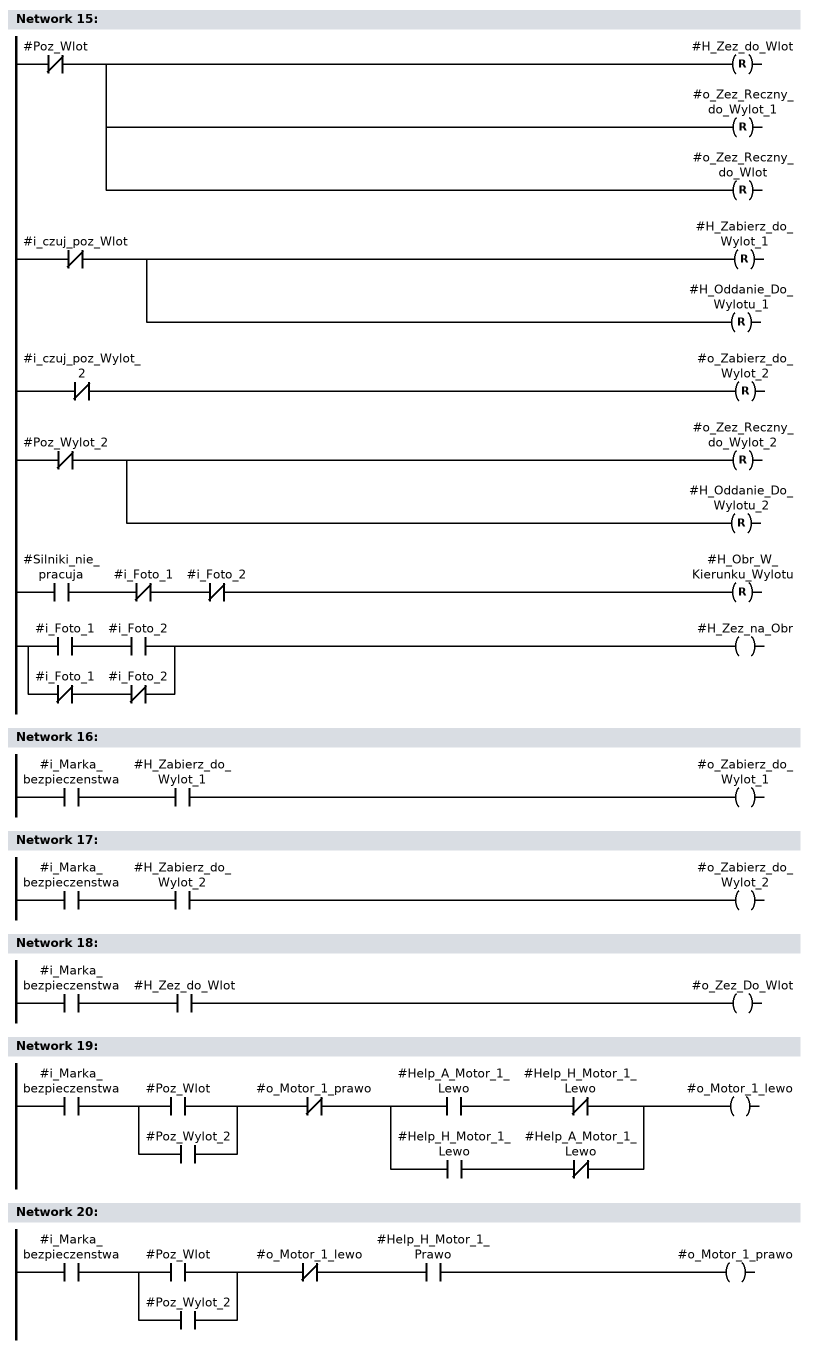
NETWORK
TITLE =
//Warunki skrajne
//
      AN    #Poz_Wlot;
      R     #H_Zez_do_Wlot;
//      R     #H_Zabierz_do_Wylot_1
      R     #o_Zez_Reczny_do_Wylot_1;
      R     #o_Zez_Reczny_do_Wlot;
      AN    #i_czuj_poz_Wlot;
      R     #H_Zabierz_do_Wylot_1;
      R     #H_Oddanie_Do_Wylotu_1;
      AN    #i_czuj_poz_Wylot_2;
      R     #o_Zabierz_do_Wylot_2;
      AN    #Poz_Wylot_2;
//      R     #o_Zabierz_do_Wylot_2
      R     #o_Zez_Reczny_do_Wylot_2;
      R     #H_Oddanie_Do_Wylotu_2;
      A     #Silniki_nie_pracuja;
      AN    #i_Foto_1;
      AN    #i_Foto_2;
      R     #H_Obr_W_Kierunku_Wylotu;
      A     #i_Foto_1;
      A     #i_Foto_2;
      O;
      AN    #i_Foto_1;
      AN    #i_Foto_2;
      =     #H_Zez_na_Obr;
NETWORK
TITLE =
//Sygnal zabierz Wylot_1
      A     #i_Marka_bezpieczenstwa;
      A     #H_Zabierz_do_Wylot_1;
      =     #o_Zabierz_do_Wylot_1;
NETWORK
TITLE =
//Sygnal zabierz Wylot_2
      A     #i_Marka_bezpieczenstwa;
      A     #H_Zabierz_do_Wylot_2;
      =     #o_Zabierz_do_Wylot_2;
NETWORK
TITLE =
//zezwolenie do porzedniej
      A     #i_Marka_bezpieczenstwa;
      A     #H_Zez_do_Wlot;
      =     #o_Zez_Do_Wlot;
NETWORK
TITLE =
////jazda automatyka reczny przod
      A     #i_Marka_bezpieczenstwa;
      A(;
      O     #Poz_Wlot;
      O     #Poz_Wylot_2;
      );
      AN    #o_Motor_1_prawo;
      A(;
      A     #Help_A_Motor_1_Lewo;
      AN    #Help_H_Motor_1_Lewo;
      O;
      A     #Help_H_Motor_1_Lewo;
      AN    #Help_A_Motor_1_Lewo;
      );
      =     #o_Motor_1_lewo;
NETWORK
TITLE =
////Jazda reczny tyl
      A     #i_Marka_bezpieczenstwa;
      A(;
      O     #Poz_Wlot;
      O     #Poz_Wylot_2;
      );
      AN    #o_Motor_1_lewo;
      A     #Help_H_Motor_1_Prawo;
      =     #o_Motor_1_prawo;
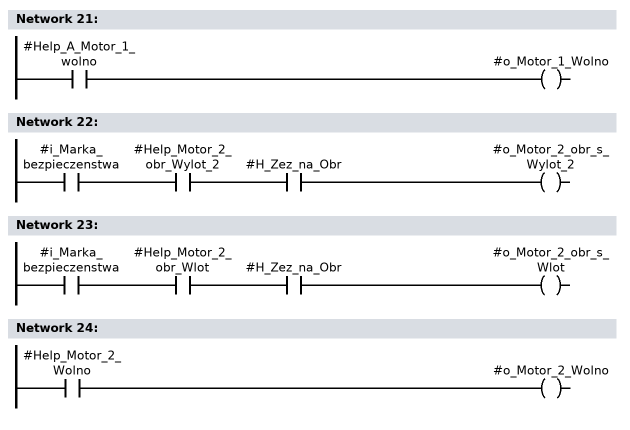
NETWORK
TITLE =
//Motor 1 wolno
      A     #Help_A_Motor_1_wolno;
      =     #o_Motor_1_Wolno;
NETWORK
TITLE =
//obrot obrotnica cc-wise
      A     #i_Marka_bezpieczenstwa;
      A     #Help_Motor_2_obr_Wylot_2;
      A     #H_Zez_na_Obr;
      =     #o_Motor_2_obr_s_Wylot_2;
NETWORK
TITLE =
//obrot obrotnica c-wise
      A     #i_Marka_bezpieczenstwa;
      A     #Help_Motor_2_obr_Wlot;
      A     #H_Zez_na_Obr;
      =     #o_Motor_2_obr_s_Wlot;
NETWORK
TITLE =
//motor 2 wolno
      A     #Help_Motor_2_Wolno;
      =     #o_Motor_2_Wolno;
END_FUNCTION_BLOCK

FUNCTION_BLOCK "Banda_Poj_+_Winda"	// FB 37
//Funkcja realizujaca koncepcje bandy pojedycznej, ktora uwzglednia rowniez tryb 
//reczny. W celu lepszego sterowania trybem recznym nalezy do³o¿yæ:
//-fotokomorki na tyle bandy.
//-fotokomorka na tyle okresla rowniez zajetosc
//-jazda do tylu bandy mozliwa
//-jazda do przodu poza fotokomorke mozliwa gdy nastepna w ruchu i wolna.
//-do³o¿enie okresnia trybu reczny/auto gdzie auto to 1 
//
//
//Do wersji z winda
//-winda rowniez aktywna gdy dojechala do gory tkz nadrabianie wysokosci
//-uwzglednione dwa czujniki od skrajnych pozycji windy
//-banda poprzedzajaca poziom 0
//-banda nastepna poziom +1
//
AUTHOR : Kng
FAMILY : Bandy
NAME : B_Single
VERSION : 0.0
VAR_INPUT
  i_Marka_Bezpieczenstwa : BOOL ;
  i_Blokada_Gdy_Uzbrajanie : BOOL ;	//Sygnal Rezerwy
  i_Auto_Reczny : BOOL ;	//1-auto,0-reczny
  i_Foto_Przod : BOOL ;	//Foto na koncu tasmy
  i_Foto_Tyl : BOOL ;	//Foto zapobiegajace wyjechaniu palety do tylu
  i_Winda_W_Gorze : BOOL ;
  i_Winda_W_Dole : BOOL ;
  i_Zez_Od_Nast : BOOL ;
  i_Paleta_Dost_Od_Nast : BOOL ;
  i_Zez_Reczny_Od_Nast : BOOL ;
  i_Zabierz_Od_Pop : BOOL ;
  i_Zez_Reczny_Od_Pop : BOOL ;
  i_PB_Jazda_Tyl : BOOL ;
  i_PB_Jazda_Przod : BOOL ;
  i_PB_Winda_Gora : BOOL ;
  i_PB_Winda_Dol : BOOL ;
  Czas_Kontroli_Przejazdu : TIME ;
END_VAR
VAR_OUTPUT
  o_Zabierz_Do_Nast : BOOL ;	//Rozkaz pobrania do nast bandy
  o_Zez_Do_Pop : BOOL ;
  o_Paleta_Dost_Do_Pop : BOOL ;
  o_Motor_Lewo : BOOL ;
  o_Motor_Prawo : BOOL ;
  o_Winda_Gora : BOOL ;
  o_Winda_Dol : BOOL ;
  o_Zez_Reczny_Do_Nast : BOOL ;
  o_Zez_Reczny_Do_Pop : BOOL ;
  o_Zajetosc_Nieb : BOOL ;	//Dla bezpieczenstwa transportu
  o_Paleta_Na_Stanowisku : BOOL ;	//Informacja o tym ze paleta jest na stanowisku
END_VAR
VAR
  Czas_kontrolny : FB 21;
  Czas_Windy : SFB 4;
  Help_A_Motor_Lewo : BOOL ;
  S_Help_Zab_Od_Pop : BOOL ;
  Stop_Czas_Kontrolny : BOOL ;
  Zbocze_1 : BOOL ;
  Zbocze_2 : BOOL ;
  Blokada_Wjazdu : BOOL ;
  Help_H_Motor_Prawo : BOOL ;
  Help_H_Motor_Lewo : BOOL ;
  Toggle : BOOL ;	//bit przemienny dla auto i hand
  H_Winda_A_Gora : BOOL ;
  H_Winda_A_Dol : BOOL ;
  H_Kontr_Windy_Gora : BOOL ;	//Kontrola by winda nie opadala
  H_Kontr_Windy_Dol : BOOL ;
  H_Winda_H_Gora : BOOL ;
  H_Winda_H_Dol : BOOL ;
  Czas_Opoz_Windy : SFB 4;
END_VAR
VAR_TEMP
  Temp_Help_1 : BOOL ;
  Temp_Help_2 : BOOL ;
  Czas_zadany : TIME ;
  Czas_aktualny : TIME ;
END_VAR
BEGIN
NETWORK
TITLE =
//
// B1        B2         foto_1    foto_2         B5        B6
//(\\\\\\\\\\\\\\\\\\)  (\\\\\\\\\\\\\\\\\\)  (\\\\\\\\\\\\\\\\\\)
//                  M1                    M2                     M3
//         
//        zabierz <-- pobierz      |  zabierz    <--  pobierz  
//     zez_do_pop --> zez_od_nast  |  zez_od_pop -->  zez_od_nast
//                                  
//-Uklad dzielony jest na realizowane funkcje
//
//         <----------------------------------------- kierunek
//                  
//
// ten network celowo jest pusty
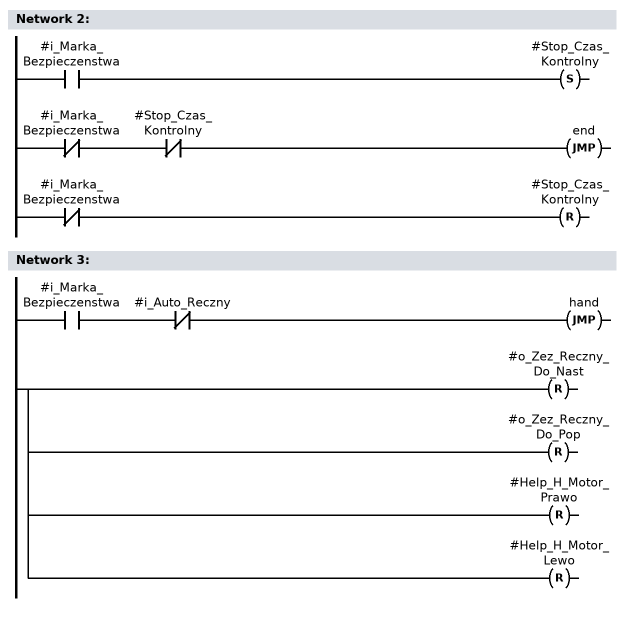
NETWORK
TITLE =
//Sprawdzenie stanu bezpieczenstwa lub freeze
//Skocz jezeli brak marki bezpieczenstwa
//Marka bezpieczenstwa ok gdy wysoki
      A     #i_Marka_Bezpieczenstwa;
      S     #Stop_Czas_Kontrolny;
      AN    #i_Marka_Bezpieczenstwa;
      AN    #Stop_Czas_Kontrolny;
      JC    end;
      AN    #i_Marka_Bezpieczenstwa;
      R     #Stop_Czas_Kontrolny;
NETWORK
TITLE =
//Wyznczenie zbocza pozytywnego i negatywnego
//skok do trybu recznego 
      A     #i_Marka_Bezpieczenstwa;
      AN    #i_Auto_Reczny;
      JC    hand;
//czyszczenie trybu recznego
      SET;
      R     #o_Zez_Reczny_Do_Nast;
      R     #o_Zez_Reczny_Do_Pop;
      R     #Help_H_Motor_Prawo;
      R     #Help_H_Motor_Lewo;
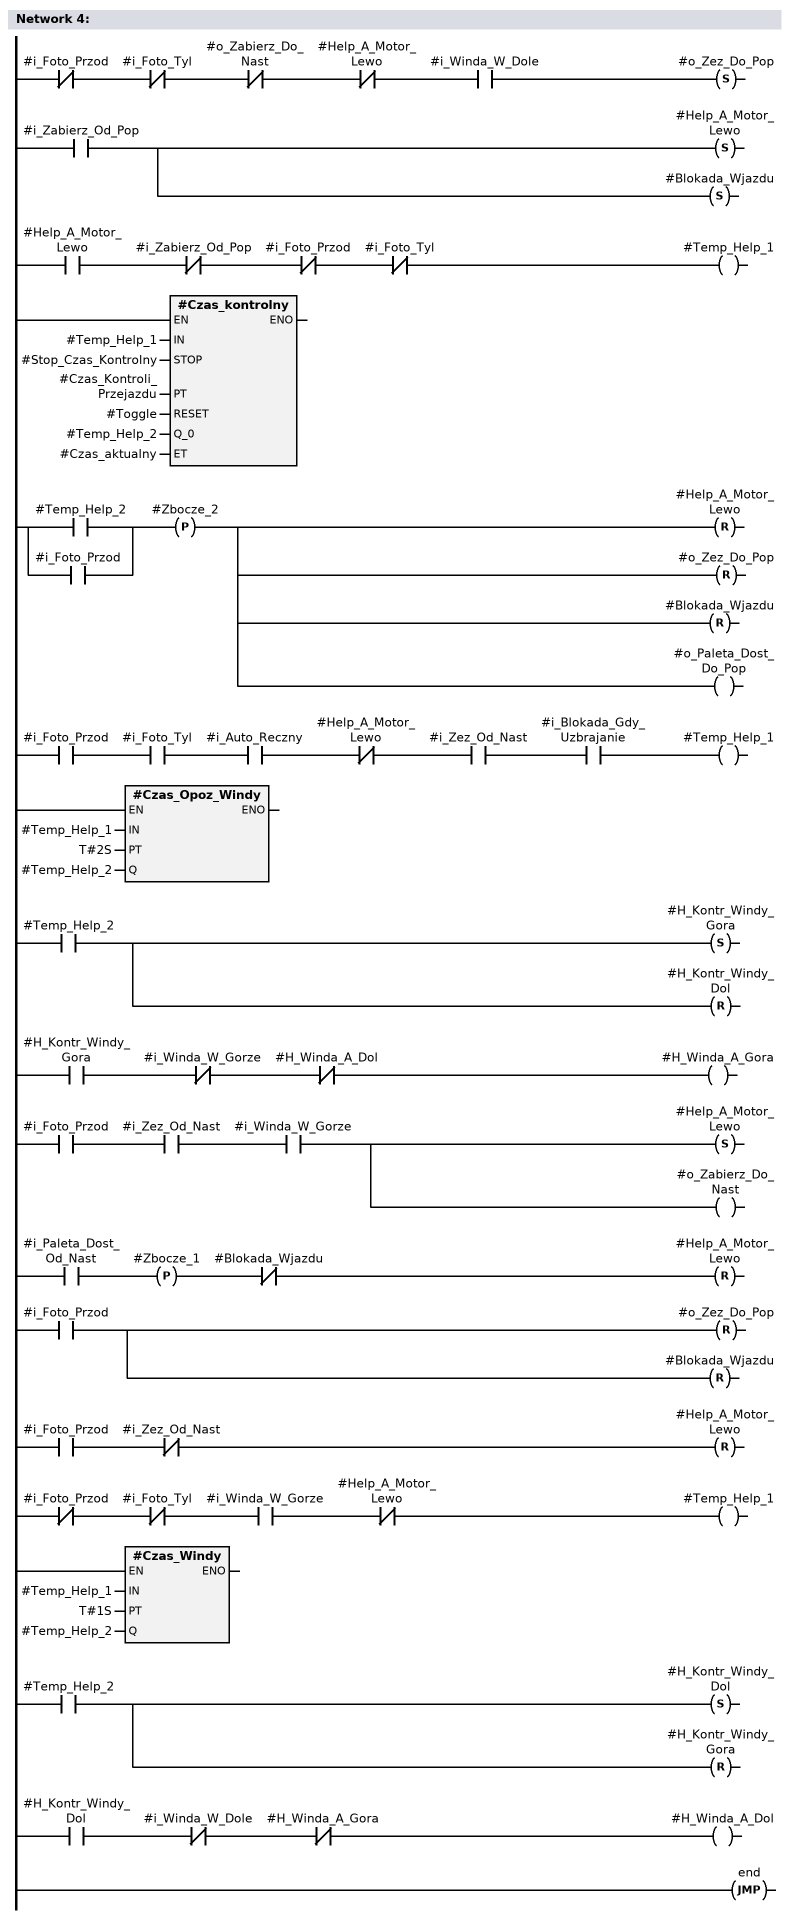
NETWORK
TITLE =
//Banda pusta zezwol na wjazd
      AN    #i_Foto_Przod;
      AN    #i_Foto_Tyl;	//dodano bo hand
      AN    #o_Zabierz_Do_Nast;
      AN    #Help_A_Motor_Lewo;
      A     #i_Winda_W_Dole;
      S     #o_Zez_Do_Pop;
      A     #i_Zabierz_Od_Pop;
      S     #Help_A_Motor_Lewo;
      S     #Blokada_Wjazdu;
//Warunek gdy pobranie z poprzedniej i miejsce foto srodek
//jest zajete
      A     #Help_A_Motor_Lewo;
      AN    #i_Zabierz_Od_Pop;
      AN    #i_Foto_Przod;
      AN    #i_Foto_Tyl;	//dodano bo hand
      =     #Temp_Help_1;
      CALL  #Czas_kontrolny (
           IN                       := #Temp_Help_1,
           STOP                     := #Stop_Czas_Kontrolny,
           PT                       := #Czas_Kontroli_Przejazdu,
           RESET                    := #Toggle,
           Q_0                      := #Temp_Help_2,
           ET                       := #Czas_aktualny);
//Paleta dostarczona
      A     #Temp_Help_2;
      O;
      A     #i_Foto_Przod;
      FP    #Zbocze_2;
      R     #Help_A_Motor_Lewo;
      R     #o_Zez_Do_Pop;
      R     #Blokada_Wjazdu;
      =     #o_Paleta_Dost_Do_Pop;
//Podniesiesnie plety na poziom +1
      A     #i_Foto_Przod;
      A     #i_Foto_Tyl;	//Aby bylo pewne pokrycie
      A     #i_Auto_Reczny;
      AN    #Help_A_Motor_Lewo;
      A     #i_Zez_Od_Nast;
      A     #i_Blokada_Gdy_Uzbrajanie;
      =     #Temp_Help_1;
      CALL  #Czas_Opoz_Windy (
           IN                       := #Temp_Help_1,
           PT                       := T#2S,
           Q                        := #Temp_Help_2);
      A     #Temp_Help_2;
      S     #H_Kontr_Windy_Gora;
      R     #H_Kontr_Windy_Dol;
      A     #H_Kontr_Windy_Gora;
//Wylaczenie windy gdy znajduje sie w gorze
      AN    #i_Winda_W_Gorze;
      AN    #H_Winda_A_Dol;
      =     #H_Winda_A_Gora;
      A     #i_Foto_Przod;
//jest zezwolenie od nastepnej
      A     #i_Zez_Od_Nast;
      A     #i_Winda_W_Gorze;
      S     #Help_A_Motor_Lewo;
      =     #o_Zabierz_Do_Nast;
      A     #i_Paleta_Dost_Od_Nast;
//Potwierdzenie otrzymania palety
      FP    #Zbocze_1;
      AN    #Blokada_Wjazdu;
      R     #Help_A_Motor_Lewo;
      A     #i_Foto_Przod;
//Gdy zajete Foto_1 brak zezwolenia do poprzedniej
      R     #o_Zez_Do_Pop;
      R     #Blokada_Wjazdu;
      A     #i_Foto_Przod;
//warunkowe zakonczenie pracy silnika gdy brak zezwolenia
//z nastepnej
      AN    #i_Zez_Od_Nast;
      R     #Help_A_Motor_Lewo;
      AN    #i_Foto_Przod;
//Powrot windy na dol
      AN    #i_Foto_Tyl;
      A     #i_Winda_W_Gorze;
      AN    #Help_A_Motor_Lewo;
      =     #Temp_Help_1;
      CALL  #Czas_Windy (
           IN                       := #Temp_Help_1,
           PT                       := T#1S,
           Q                        := #Temp_Help_2);
      A     #Temp_Help_2;
      S     #H_Kontr_Windy_Dol;
      R     #H_Kontr_Windy_Gora;
      A     #H_Kontr_Windy_Dol;
      AN    #i_Winda_W_Dole;
      AN    #H_Winda_A_Gora;
      =     #H_Winda_A_Dol;
      JU    end;
//skocz do koniec
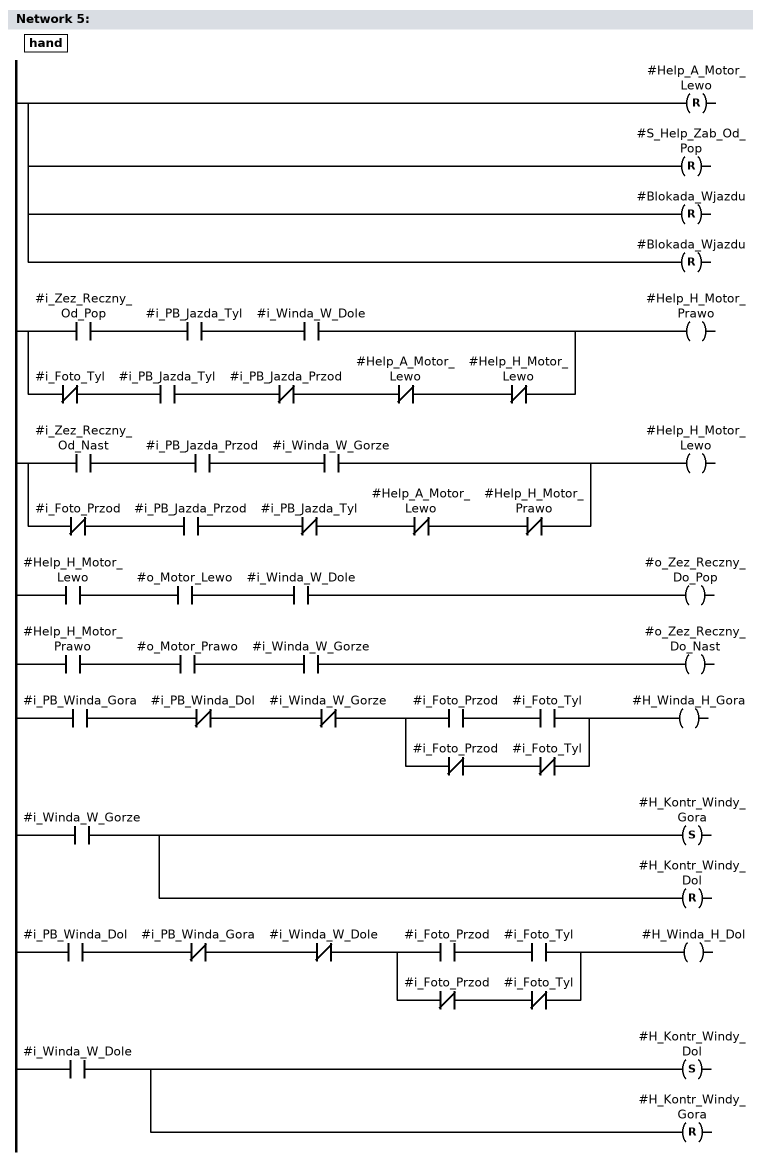
NETWORK
TITLE =
//Tryb reczny
//
hand: NOP   0;
//czyszczenie bitow z automatyki
      SET;
      R     #Help_A_Motor_Lewo;
      R     #S_Help_Zab_Od_Pop;
      R     #Blokada_Wjazdu;
      R     #Blokada_Wjazdu;
//ustawienie przyciskow
//jazda do tylu przycisk tyl
      A     #i_Zez_Reczny_Od_Pop;
      A     #i_PB_Jazda_Tyl;
      A     #i_Winda_W_Dole;
      O;
      AN    #i_Foto_Tyl;
      A(;
      A     #i_PB_Jazda_Tyl;
      AN    #i_PB_Jazda_Przod;
      AN    #Help_A_Motor_Lewo;
      AN    #Help_H_Motor_Lewo;
      );
      =     #Help_H_Motor_Prawo;
//jazda do przodu
      A     #i_Zez_Reczny_Od_Nast;
      A     #i_PB_Jazda_Przod;
      A     #i_Winda_W_Gorze;
      O;
      AN    #i_Foto_Przod;
      A(;
      A     #i_PB_Jazda_Przod;
      AN    #i_PB_Jazda_Tyl;
      AN    #Help_A_Motor_Lewo;
      AN    #Help_H_Motor_Prawo;
      );
      =     #Help_H_Motor_Lewo;
//zezwolenie do poprzedniej
      A     #Help_H_Motor_Lewo;
      A     #o_Motor_Lewo;
      A     #i_Winda_W_Dole;
      =     #o_Zez_Reczny_Do_Pop;
//zezwolenie do nastepnej
      A     #Help_H_Motor_Prawo;
      A     #o_Motor_Prawo;
      A     #i_Winda_W_Gorze;
      =     #o_Zez_Reczny_Do_Nast;
//Jazda windy   gora
      A     #i_PB_Winda_Gora;
      AN    #i_PB_Winda_Dol;
      AN    #i_Winda_W_Gorze;
      A(;
      A     #i_Foto_Przod;
      A     #i_Foto_Tyl;
      O;
      AN    #i_Foto_Przod;
      AN    #i_Foto_Tyl;
      );
      =     #H_Winda_H_Gora;
      A     #i_Winda_W_Gorze;
      S     #H_Kontr_Windy_Gora;
      R     #H_Kontr_Windy_Dol;
//Jazda Windy dol
      A     #i_PB_Winda_Dol;
      AN    #i_PB_Winda_Gora;
      AN    #i_Winda_W_Dole;
      A(;
      A     #i_Foto_Przod;
      A     #i_Foto_Tyl;
      O;
      AN    #i_Foto_Przod;
      AN    #i_Foto_Tyl;
      );
      =     #H_Winda_H_Dol;
      A     #i_Winda_W_Dole;
      S     #H_Kontr_Windy_Dol;
      R     #H_Kontr_Windy_Gora;
NETWORK
TITLE =
//Przypisanie wyjsc
//Koniec skoku
end:  NOP   0;
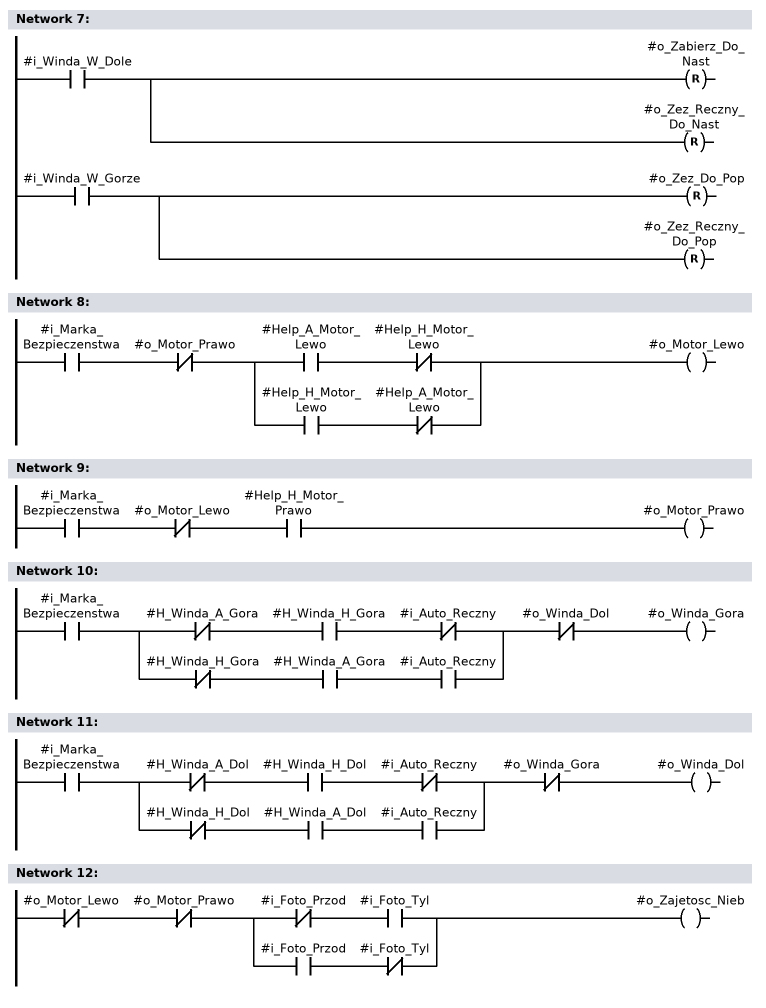
NETWORK
TITLE =
//warunki skrajne
//
      A     #i_Winda_W_Dole;
      R     #o_Zabierz_Do_Nast;
      R     #o_Zez_Reczny_Do_Nast;
      A     #i_Winda_W_Gorze;
      R     #o_Zez_Do_Pop;
      R     #o_Zez_Reczny_Do_Pop;
NETWORK
TITLE =
////jazda automatyka reczny przod
      A     #i_Marka_Bezpieczenstwa;
      AN    #o_Motor_Prawo;
      A(;
      A     #Help_A_Motor_Lewo;
      AN    #Help_H_Motor_Lewo;
      O;
      A     #Help_H_Motor_Lewo;
      AN    #Help_A_Motor_Lewo;
      );
      =     #o_Motor_Lewo;
NETWORK
TITLE =
////Jazda reczny tyl
      A     #i_Marka_Bezpieczenstwa;
      AN    #o_Motor_Lewo;
      A     #Help_H_Motor_Prawo;
      =     #o_Motor_Prawo;
NETWORK
TITLE =
//winda gora
//
      A     #i_Marka_Bezpieczenstwa;
      A(;
      AN    #H_Winda_A_Gora;
      A     #H_Winda_H_Gora;
      AN    #i_Auto_Reczny;
      O;
      AN    #H_Winda_H_Gora;
      A     #H_Winda_A_Gora;
      A     #i_Auto_Reczny;
      );
      AN    #o_Winda_Dol;
      =     #o_Winda_Gora;
NETWORK
TITLE =
//winda dol
      A     #i_Marka_Bezpieczenstwa;
      A(;
      AN    #H_Winda_A_Dol;
      A     #H_Winda_H_Dol;
      AN    #i_Auto_Reczny;
      O;
      AN    #H_Winda_H_Dol;
      A     #H_Winda_A_Dol;
      A     #i_Auto_Reczny;
      );
      AN    #o_Winda_Gora;
      =     #o_Winda_Dol;
NETWORK
TITLE =
//Zajetosc
      AN    #o_Motor_Lewo;
      AN    #o_Motor_Prawo;
      A(;
      AN    #i_Foto_Przod;
      A     #i_Foto_Tyl;
      O;
      A     #i_Foto_Przod;
      AN    #i_Foto_Tyl;
      );
      =     #o_Zajetosc_Nieb;
NETWORK
TITLE =
//Koniec
//koniec
      BEU;
END_FUNCTION_BLOCK

FUNCTION_BLOCK "Obr_Na_Poz_1_Pelny"	// FB 61
AUTHOR : Kng
NAME : B_Obr
VERSION : 0.1
VAR_INPUT
  i_Auto_Reczny : BOOL ;
  i_Tryb_Uzbrajanie : BOOL ;	//Tryb uzbrajania palaty (mozliwosci pelnego obrotu)
  i_Obracaj_W_Lewo : BOOL ;	//Aktywne tylko w trybie uzbrajania
  i_Obracaj_W_Prawo : BOOL ;	//Aktywne tylko w trybie uzbrajania
  i_Jedz_Na_0st : BOOL ;
  i_Jedz_Na_90st : BOOL ;
  i_Czujnik_0st : BOOL ;
  i_Czujnik_90st : BOOL ;
  i_Czujnik_Ham_0st : BOOL ;
  i_Czujnik_Ham_90st : BOOL ;
  i_Odblokuj_Obrotnice : BOOL ;
END_VAR
VAR_OUTPUT
  o_Na_Pozycji_0st : BOOL ;	//Obrotnica na pozycji 0 stopni
  o_Na_Pozycji_90st : BOOL ;	//Obrotnica na pozycji 90 stopni
  o_Motor_Wolno : BOOL ;
  o_Odblokowanie_Rolek : BOOL ;
  o_Uzbrajanie : BOOL ;
END_VAR
VAR_IN_OUT
  io_Talerz_w_Lewo : BOOL ;
  io_Talerz_w_Prawo : BOOL ;
END_VAR
VAR
  Czas_Dojscia : SFB 4;
  Czas_Startu : SFB 4;
  Help_Start : BOOL ;
  H_Blokada_Uzbrajania : BOOL ;
  H_2 : BOOL ;
  H_3 : BOOL ;
  H_4 : BOOL ;
END_VAR
VAR_TEMP
  Help_1 : BOOL ;
END_VAR
BEGIN
NETWORK
TITLE =
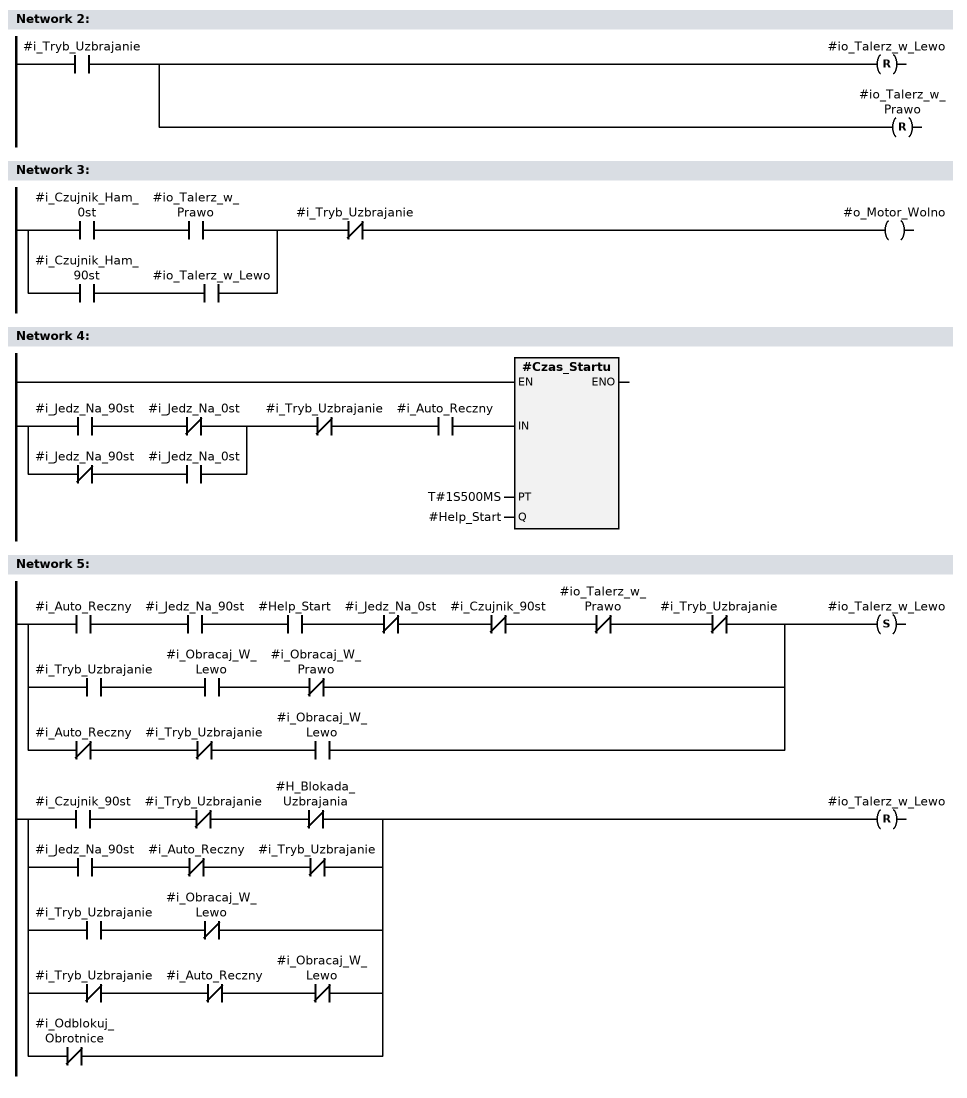
NETWORK
TITLE =
//Tryb uzbrajania resetuje wszystkie bity
      A     #i_Tryb_Uzbrajanie;
      R     #io_Talerz_w_Lewo;
      R     #io_Talerz_w_Prawo;
NETWORK
TITLE =
//Motor wolno gdy czujniki hamowania
      A(;
      A     #i_Czujnik_Ham_0st;
      A     #io_Talerz_w_Prawo;
      O;
      A     #i_Czujnik_Ham_90st;
      A     #io_Talerz_w_Lewo;
      );
      AN    #i_Tryb_Uzbrajanie;
      =     #o_Motor_Wolno;
NETWORK
TITLE =
      A(;
      A     #i_Jedz_Na_90st;
      AN    #i_Jedz_Na_0st;
      O;
      AN    #i_Jedz_Na_90st;
      A     #i_Jedz_Na_0st;
      );
      AN    #i_Tryb_Uzbrajanie;
      A     #i_Auto_Reczny;
      =     L 1.0;
      BLD   103;
      CALL  #Czas_Startu (
           IN                       := L 1.0,
           PT                       := T#1S500MS,
           Q                        := #Help_Start);
      NOP   0;
NETWORK
TITLE =
      A(;
      A     #i_Auto_Reczny;
      A     #i_Jedz_Na_90st;
      A     #Help_Start;
      AN    #i_Jedz_Na_0st;
      AN    #i_Czujnik_90st;
      AN    #io_Talerz_w_Prawo;
      AN    #i_Tryb_Uzbrajanie;
      O;
      A     #i_Tryb_Uzbrajanie;
      A     #i_Obracaj_W_Lewo;
      AN    #i_Obracaj_W_Prawo;
      O;
      AN    #i_Auto_Reczny;
      AN    #i_Tryb_Uzbrajanie;
      A     #i_Obracaj_W_Lewo;
      );
      S     #io_Talerz_w_Lewo;
      A(;
      A     #i_Czujnik_90st;
      AN    #i_Tryb_Uzbrajanie;
      AN    #H_Blokada_Uzbrajania;
      O;
      A     #i_Jedz_Na_90st;
      AN    #i_Auto_Reczny;
      AN    #i_Tryb_Uzbrajanie;
      O;
      A     #i_Tryb_Uzbrajanie;
      AN    #i_Obracaj_W_Lewo;
      O;
      AN    #i_Tryb_Uzbrajanie;
      AN    #i_Auto_Reczny;
      AN    #i_Obracaj_W_Lewo;
      ON    #i_Odblokuj_Obrotnice;
      );
      R     #io_Talerz_w_Lewo;
      NOP   0;
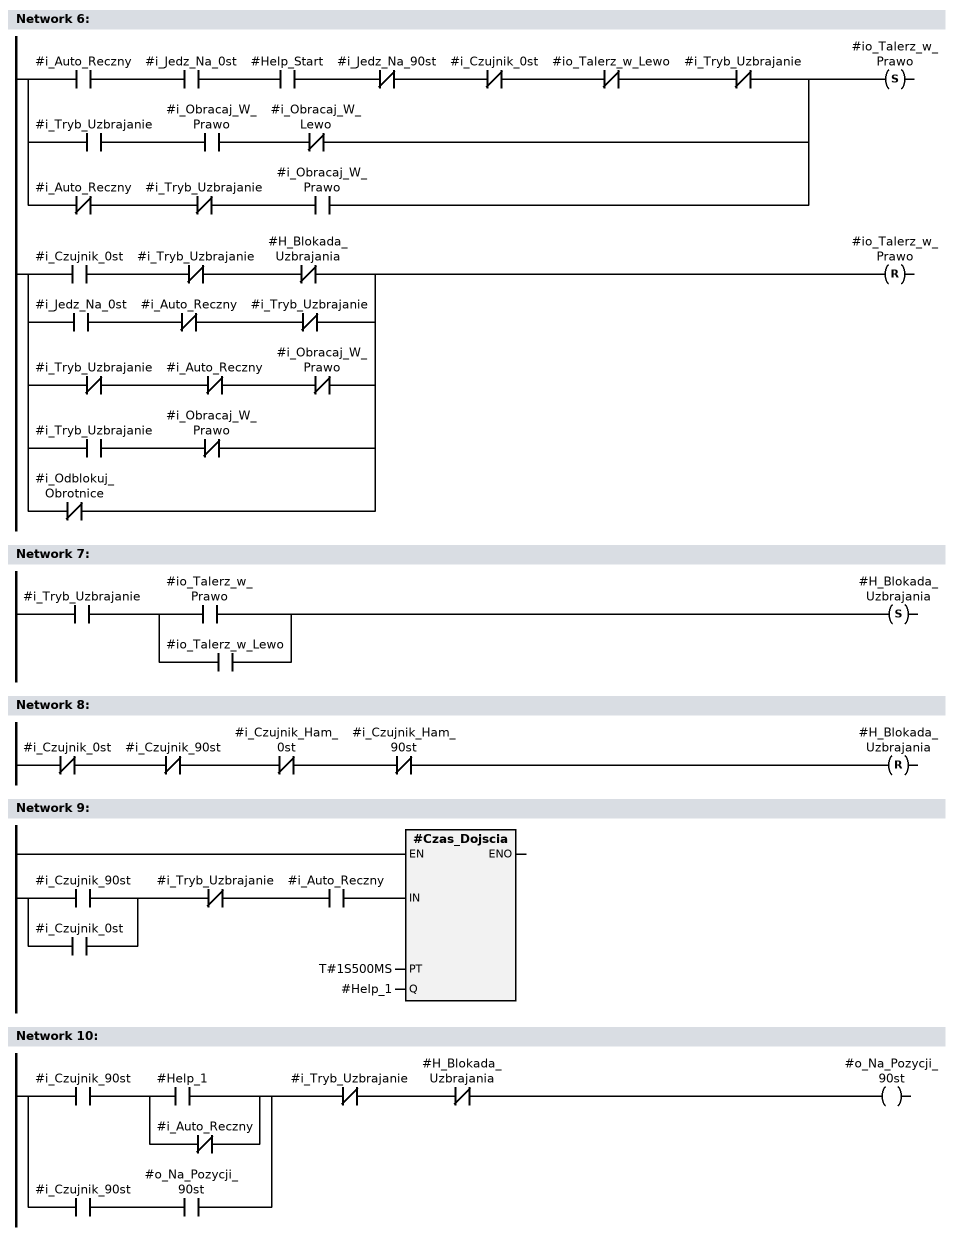
NETWORK
TITLE =
      A(;
      A     #i_Auto_Reczny;
      A     #i_Jedz_Na_0st;
      A     #Help_Start;
      AN    #i_Jedz_Na_90st;
      AN    #i_Czujnik_0st;
      AN    #io_Talerz_w_Lewo;
      AN    #i_Tryb_Uzbrajanie;
      O;
      A     #i_Tryb_Uzbrajanie;
      A     #i_Obracaj_W_Prawo;
      AN    #i_Obracaj_W_Lewo;
      O;
      AN    #i_Auto_Reczny;
      AN    #i_Tryb_Uzbrajanie;
      A     #i_Obracaj_W_Prawo;
      );
      S     #io_Talerz_w_Prawo;
      A(;
      A     #i_Czujnik_0st;
      AN    #i_Tryb_Uzbrajanie;
      AN    #H_Blokada_Uzbrajania;
      O;
      A     #i_Jedz_Na_0st;
      AN    #i_Auto_Reczny;
      AN    #i_Tryb_Uzbrajanie;
      O;
      AN    #i_Tryb_Uzbrajanie;
      AN    #i_Auto_Reczny;
      AN    #i_Obracaj_W_Prawo;
      O;
      A     #i_Tryb_Uzbrajanie;
      AN    #i_Obracaj_W_Prawo;
      ON    #i_Odblokuj_Obrotnice;
      );
      R     #io_Talerz_w_Prawo;
      NOP   0;
NETWORK
TITLE =
//Jezeli byl tryb uzbrajania aktywny i nastapil przejazd aktywuj h_1
      A     #i_Tryb_Uzbrajanie;
      A(;
      O     #io_Talerz_w_Prawo;
      O     #io_Talerz_w_Lewo;
      );
      S     #H_Blokada_Uzbrajania;
NETWORK
TITLE =
//Reset blokady uzbrajania
      AN    #i_Czujnik_0st;
      AN    #i_Czujnik_90st;
      AN    #i_Czujnik_Ham_0st;
      AN    #i_Czujnik_Ham_90st;
      R     #H_Blokada_Uzbrajania;
NETWORK
TITLE =
      A(;
      O     #i_Czujnik_90st;
      O     #i_Czujnik_0st;
      );
      AN    #i_Tryb_Uzbrajanie;
      A     #i_Auto_Reczny;
      =     L 1.0;
      BLD   103;
      CALL  #Czas_Dojscia (
           IN                       := L 1.0,
           PT                       := T#1S500MS,
           Q                        := #Help_1);
      NOP   0;
NETWORK
TITLE =
      A(;
      A     #i_Czujnik_90st;
      A(;
      O     #Help_1;
      ON    #i_Auto_Reczny;
      );
      O;
      A     #i_Czujnik_90st;
      A     #o_Na_Pozycji_90st;
      );
      AN    #i_Tryb_Uzbrajanie;
      AN    #H_Blokada_Uzbrajania;
      =     #o_Na_Pozycji_90st;
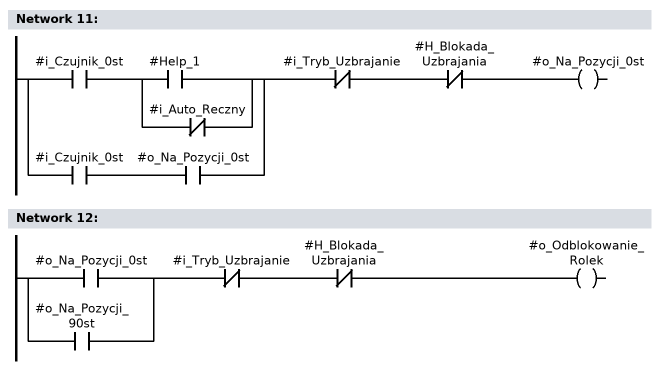
NETWORK
TITLE =
      A(;
      A     #i_Czujnik_0st;
      A(;
      O     #Help_1;
      ON    #i_Auto_Reczny;
      );
      O;
      A     #i_Czujnik_0st;
      A     #o_Na_Pozycji_0st;
      );
      AN    #i_Tryb_Uzbrajanie;
      AN    #H_Blokada_Uzbrajania;
      =     #o_Na_Pozycji_0st;
NETWORK
TITLE =
//Odblokowanie napedu rolkowego
      A(;
      O     #o_Na_Pozycji_0st;
      O     #o_Na_Pozycji_90st;
      );
      AN    #i_Tryb_Uzbrajanie;
      AN    #H_Blokada_Uzbrajania;
      =     #o_Odblokowanie_Rolek;
END_FUNCTION_BLOCK

FUNCTION "Funkcja_Bezpieczenstwa" : VOID	// FC 3
VERSION : 0.1
VAR_TEMP
  Temp_Help_1 : BOOL ;
  Temp_Help_2 : BOOL ;
END_VAR
BEGIN
NETWORK
TITLE =
//Ten network celowo jest wolny
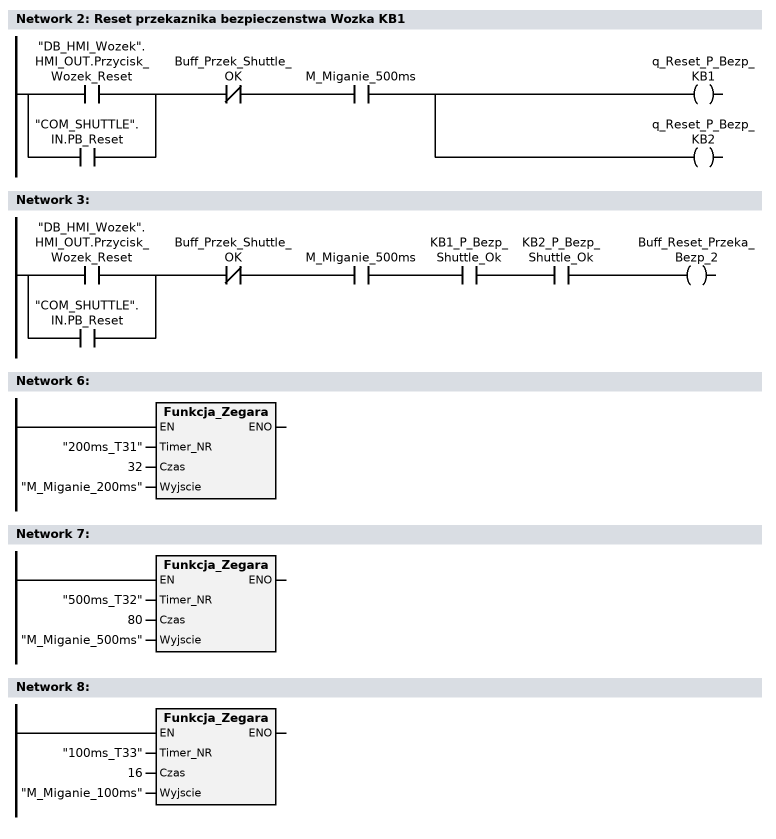
NETWORK
TITLE = Reset przekaznika bezpieczenstwa Wozka KB1
//Reset przekaznikow bezpieczenstwa stanowisk KB1,KB2
      A(;
      O     "DB_HMI_Wozek".HMI_OUT.Przycisk_Wozek_Reset;
      O     "COM_SHUTTLE".IN.PB_Reset;
      );
      AN    "Buff_Przek_Shuttle_OK";
      A     "M_Miganie_500ms";
      =     "q_Reset_P_Bezp_KB1";
      =     "q_Reset_P_Bezp_KB2";
NETWORK
TITLE =
//Reset przekaznik bezpieczenstwa wozek
      A(;
      O     "DB_HMI_Wozek".HMI_OUT.Przycisk_Wozek_Reset;
      O     "COM_SHUTTLE".IN.PB_Reset;
      );
      AN    "Buff_Przek_Shuttle_OK";
      A     "M_Miganie_500ms";
      A     "KB1_P_Bezp_Shuttle_Ok";
      A     "KB2_P_Bezp_Shuttle_Ok";
      =     "Buff_Reset_Przeka_Bezp_2";
NETWORK
TITLE =
NETWORK
TITLE =
//Zalaczenie szynoprzewodu
      A     "i_Buff_PB_Zal_Wozka";
      L     S5T#1S;
      SD    "Buff_T35";
//----
      A     "Buff_T35";
      FP    "Help_M302.7";
      X     "q_Buff_Zal_Wozka";
      =     "q_Buff_Zal_Wozka";
NETWORK
TITLE =
//Timmer generujacy takt 200ms
//
      CALL  "Funkcja_Zegara" (
           Timer_NR                 := "200ms_T31",
           Czas                     := 32,
           Wyjscie                  := "M_Miganie_200ms");
      NOP   0;
NETWORK
TITLE =
//Timmer generujacy takt 500ms
      CALL  "Funkcja_Zegara" (
           Timer_NR                 := "500ms_T32",
           Czas                     := 80,
           Wyjscie                  := "M_Miganie_500ms");
      NOP   0;
NETWORK
TITLE =
//Timmer generujacy takt 100ms
      CALL  "Funkcja_Zegara" (
           Timer_NR                 := "100ms_T33",
           Czas                     := 16,
           Wyjscie                  := "M_Miganie_100ms");
      NOP   0;
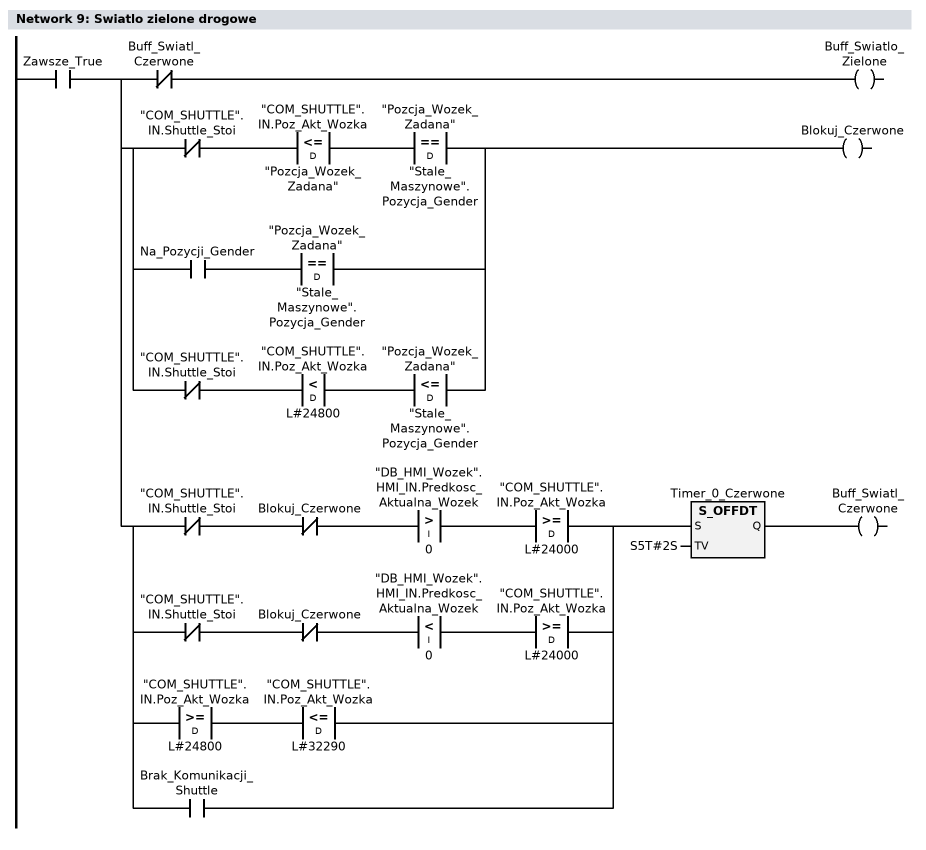
NETWORK
TITLE = Swiatlo zielone drogowe
//Ruch drogowy
//0______24000
//0______26300
//26200__32290
      A     "Zawsze_True";
      =     L 1.0;
      A     L 1.0;
      AN    "Buff_Swiatl_Czerwone";
      =     "Buff_Swiatlo_Zielone";
      A     L 1.0;
      A(;
      AN    "COM_SHUTTLE".IN.Shuttle_Stoi;
      A(;
      L     "COM_SHUTTLE".IN.Poz_Akt_Wozka;
      L     "Pozcja_Wozek_Zadana";
      <=D;
      );
      A(;
      L     "Pozcja_Wozek_Zadana";
      L     "Stale_Maszynowe".Pozycja_Gender;
      ==D;
      );
      O;
      A     "Na_Pozycji_Gender";
      A(;
      L     "Pozcja_Wozek_Zadana";
      L     "Stale_Maszynowe".Pozycja_Gender;
      ==D;
      );
      O;
      AN    "COM_SHUTTLE".IN.Shuttle_Stoi;
      A(;
      L     "COM_SHUTTLE".IN.Poz_Akt_Wozka;
      L     L#24800;
      <D;
      );
      A(;
      L     "Pozcja_Wozek_Zadana";
      L     "Stale_Maszynowe".Pozycja_Gender;
      <=D;
      );
      );
      =     "Blokuj_Czerwone";
      A     L 1.0;
      A(;
      AN    "COM_SHUTTLE".IN.Shuttle_Stoi;
      AN    "Blokuj_Czerwone";
      A(;
      L     "DB_HMI_Wozek".HMI_IN.Predkosc_Aktualna_Wozek;
      L     0;
      >I;
      );
      A(;
      L     "COM_SHUTTLE".IN.Poz_Akt_Wozka;
      L     L#24000;
      >=D;
      );
      O;
      AN    "COM_SHUTTLE".IN.Shuttle_Stoi;
      AN    "Blokuj_Czerwone";
      A(;
      L     "DB_HMI_Wozek".HMI_IN.Predkosc_Aktualna_Wozek;
      L     0;
      <I;
      );
      A(;
      L     "COM_SHUTTLE".IN.Poz_Akt_Wozka;
      L     L#24000;
      >=D;
      );
      O;
      A(;
      L     "COM_SHUTTLE".IN.Poz_Akt_Wozka;
      L     L#24800;
      >=D;
      );
      A(;
      L     "COM_SHUTTLE".IN.Poz_Akt_Wozka;
      L     L#32290;
      <=D;
      );
      O     "Brak_Komunikacji_Shuttle";
      );
      L     S5T#2S;
      SF    "Timer_0_Czerwone";
      NOP   0;
      NOP   0;
      NOP   0;
      A     "Timer_0_Czerwone";
      =     "Buff_Swiatl_Czerwone";
END_FUNCTION

FUNCTION "Wozek_Jezdny_Jazda_2" : VOID	// FC 6
//Funkcja odpowiada za sterowanie ruchem wozka. Uzywa marek od m600.0
AUTHOR : Kng
NAME : Main
VERSION : 0.1
BEGIN
NETWORK
TITLE =
//Ten Network Celowo jest wolny
NETWORK
TITLE =
      CALL  "Wozek_Jezdny_Kolejka";
      NOP   0;
NETWORK
TITLE =
//Sprawdzenie okna dla KB2
      CALL  "Sprawdzenie_Okna" (
           War_Pozycji_Aktualnej    := "COM_SHUTTLE".IN.Poz_Akt_Wozka,
           War_Pozycji_Zadanej      := "COM_SHUTTLE".OUT.Pozycja_Zadana,
           War_Pozycji_Maszyn       := "Stale_Maszynowe".Pozycja_KB1,
           Tolerancja               := L#30,
           Na_Pozycji_Maszyny       := "Marka_X",
           Na_Pozycji_Zadanej       := "Marka_X",
           Na_Poz_Zad_Masz          := "Na_Pozycji_KB1");
      CALL  "Sprawdzenie_Okna" (
           War_Pozycji_Aktualnej    := "COM_SHUTTLE".IN.Poz_Akt_Wozka,
           War_Pozycji_Zadanej      := "COM_SHUTTLE".OUT.Pozycja_Zadana,
           War_Pozycji_Maszyn       := "Stale_Maszynowe".Pozycja_KB2,
           Tolerancja               := L#30,
           Na_Pozycji_Maszyny       := "Marka_X",
           Na_Pozycji_Zadanej       := "Marka_X",
           Na_Poz_Zad_Masz          := "Na_Pozycji_KB2");
      CALL  "Sprawdzenie_Okna" (
           War_Pozycji_Aktualnej    := "COM_SHUTTLE".IN.Poz_Akt_Wozka,
           War_Pozycji_Zadanej      := "COM_SHUTTLE".OUT.Pozycja_Zadana,
           War_Pozycji_Maszyn       := "Stale_Maszynowe".Pozycja_Gender,
           Tolerancja               := L#20,
           Na_Pozycji_Maszyny       := "Marka_X",
           Na_Pozycji_Zadanej       := "Marka_X",
           Na_Poz_Zad_Masz          := "Na_Pozycji_Gender");
      CALL  "Sprawdzenie_Okna" (
           War_Pozycji_Aktualnej    := "COM_SHUTTLE".IN.Poz_Akt_Wozka,
           War_Pozycji_Zadanej      := "COM_SHUTTLE".OUT.Pozycja_Zadana,
           War_Pozycji_Maszyn       := "Stale_Maszynowe".Pozycja_odbieranie,
           Tolerancja               := L#20,
           Na_Pozycji_Maszyny       := "Marka_X",
           Na_Pozycji_Zadanej       := "Marka_X",
           Na_Poz_Zad_Masz          := "Na_Pozycji_Odbieranie");
NETWORK
TITLE =
//Pozycja Intro pobieranie
      CALL  "Sprawdzenie_Okna" (
           War_Pozycji_Aktualnej    := "COM_SHUTTLE".IN.Poz_Akt_Wozka,
           War_Pozycji_Zadanej      := "COM_SHUTTLE".OUT.Pozycja_Zadana,
           War_Pozycji_Maszyn       := "Stale_Maszynowe".Pozycja_Pob_I1,
           Tolerancja               := L#20,
           Na_Pozycji_Maszyny       := "Marka_X",
           Na_Pozycji_Zadanej       := "Marka_X",
           Na_Poz_Zad_Masz          := "Na_Pozycji_Pob_I1");
      CALL  "Sprawdzenie_Okna" (
           War_Pozycji_Aktualnej    := "COM_SHUTTLE".IN.Poz_Akt_Wozka,
           War_Pozycji_Zadanej      := "COM_SHUTTLE".OUT.Pozycja_Zadana,
           War_Pozycji_Maszyn       := "Stale_Maszynowe".Pozycja_Pob_I2,
           Tolerancja               := L#20,
           Na_Pozycji_Maszyny       := "Marka_X",
           Na_Pozycji_Zadanej       := "Marka_X",
           Na_Poz_Zad_Masz          := "Na_Pozycji_Pob_I2");
      CALL  "Sprawdzenie_Okna" (
           War_Pozycji_Aktualnej    := "COM_SHUTTLE".IN.Poz_Akt_Wozka,
           War_Pozycji_Zadanej      := "COM_SHUTTLE".OUT.Pozycja_Zadana,
           War_Pozycji_Maszyn       := "Stale_Maszynowe".Pozycja_Pob_I3,
           Tolerancja               := L#20,
           Na_Pozycji_Maszyny       := "Marka_X",
           Na_Pozycji_Zadanej       := "Marka_X",
           Na_Poz_Zad_Masz          := "Na_Pozycji_Pob_I3");
NETWORK
TITLE =
//Warunki zasprzeglenia 
      A     "Zawsze_True";
      =     L 0.0;
      A(;
      A     L 0.0;
      A     "KB1_Auto_Reczny";
      FN    "Edge_M606.0";
      );
      A     "Zasprzeglenie_KB1";
      =     "KB1_Przej_Auto_Na_Recz";
      A(;
      A     L 0.0;
      A     "COM_SHUTTLE".IN.Shuttle_Stoi;
      FP    "Edge_M608.0";
      );
      A     "Na_Pozycji_KB1";
      AN    "KB1_Auto_Reczny";
      AN    "DB_HMI_Wozek".HMI_IN.Wozek_W_Trybie_Auto;
      AN    "Zasprzeglenie_KB1";
      =     "Warunk_Zasprz_KB1";
      A(;
      A     L 0.0;
      A     "KB2_Auto_Reczny";
      FN    "Edge_M606.1";
      );
      A     "Zasprzeglenie_KB2";
      =     "KB2_Przej_Auto_Na_Recz";
      A(;
      A     L 0.0;
      A     "COM_SHUTTLE".IN.Shuttle_Stoi;
      FP    "Edge_M608.1";
      );
      A     "Na_Pozycji_KB2";
      AN    "KB2_Auto_Reczny";
      AN    "DB_HMI_Wozek".HMI_IN.Wozek_W_Trybie_Auto;
      AN    "Zasprzeglenie_KB2";
      =     "Warunk_Zasprz_KB2";
NETWORK
TITLE =
//Buffory
      A     "Zawsze_True";
      =     L 0.0;
      A(;
      A     L 0.0;
      A(;
      O     "I1_Buf_Auto_Reczny";
      O     "I2_I3_Buf_Auto_Reczny";
      );
      FN    "Edge_M606.2";
      );
      A(;
      O     "Zasprzeglenie_Pob_I1";
      O     "Zasprzeglenie_Odbieranie";
      );
      =     "Buff_Przejscie_Na_Recz";
      A(;
      A     L 0.0;
      A     "COM_SHUTTLE".IN.Shuttle_Stoi;
      FP    "Edge_M608.2";
      );
      A(;
      O     "Na_Pozycji_Odbieranie";
      O     "Na_Pozycji_Pob_I1";
      O     "Na_Pozycji_Pob_I2";
      O     "Na_Pozycji_Pob_I3";
      );
      AN    "I1_Buf_Auto_Reczny";
      AN    "DB_HMI_Wozek".HMI_IN.Wozek_W_Trybie_Auto;
      =     M 606.4;
      A     L 0.0;
      A     M 606.4;
      AN    "Zasprzeglenie_Odbieranie";
      AN    "Zasprzeglenie_Pob_I1";
      AN    "Zasprzeglenie_Pob_I2";
      AN    "Zasprzeglenie_Pob_I3";
      =     "Warunk_Zasprz_Buffory";
NETWORK
TITLE =
//Gender
      A     "Zawsze_True";
      =     L 0.0;
      A(;
      A     L 0.0;
      A     "Gender_Auto_Reczny";
      FN    "Edge_M606.3";
      );
      A     "Zasprzeglenie_Gender";
      =     "Gen_Przejscie_Na_Reczny";
      A(;
      A     L 0.0;
      A     "COM_SHUTTLE".IN.Shuttle_Stoi;
      FP    "Edge_M608.3";
      );
      A     "Na_Pozycji_Gender";
      AN    "Gender_Auto_Reczny";
      AN    "DB_HMI_Wozek".HMI_IN.Wozek_W_Trybie_Auto;
      AN    "Zasprzeglenie_Gender";
      =     "Warunk_Zasprz_Gender";
NETWORK
TITLE = Wozek zasprzeglony do KB1
//Zasprzeglenie wozka w trybie recznym .Polaczone z funkcja FB8 
////KB1
      A     "Na_Pozycji_KB1";
      =     L 0.0;
      A     L 0.0;
      A     "KB1_Auto_Reczny";
      A     "Przejmij_Z_KB1";
      AN    "Marka_Jazdy_Na_Nowa_Poz";
      S     "Zasprzeglenie_KB1";
      A     L 0.0;
      A(;
      AN    "KB1_Auto_Reczny";
      A     "KB1_PB_Semi_Auto";
      O     "KB1_Przej_Auto_Na_Recz";
      O     "Warunk_Zasprz_KB1";
      );
      AN    "Marka_Jazdy_Na_Nowa_Poz";
      S     "Wozek_Na_Reczny";
      R     "Wozek_Na_Auto";
      S     "Zasprzeglenie_KB1";
      R     "Marka_Jazdy_Na_Nowa_Poz";
      A(;
      A     L 0.0;
      A     "KB1_Auto_Reczny";
      A     "KB1_PB_Auto";
      L     S5T#1S;
      SD    "Timmer_102_KB1";
      NOP   0;
      NOP   0;
      NOP   0;
      A     "Timmer_102_KB1";
      );
      AN    "Marka_Jazdy_Na_Nowa_Poz";
      =     L 0.1;
      A     L 0.1;
      BLD   102;
      S     "Wozek_Na_Auto";
      A     L 0.1;
      BLD   102;
      R     "Wozek_Na_Reczny";
      A     L 0.1;
      AN    "DB_CONECTOR_KB1".Winda.Foto_2;
      AN    "Foto_Pokryte_Czasowo";
      R     "Zasprzeglenie_KB1";
NETWORK
TITLE = Wozek zasprzeglony do KB1
//Przejmij kod kolbusa 1
////KB1
      A     "Zasprzeglenie_KB1";
      A(;
      A     "KB1_Auto_Reczny";
      A     "Na_Pozycji_KB1";
      A     "Foto_Wozek_Przod";
      A     "Foto_Wozek_Tyl";
      A     "Foto_Pokryte_Czasowo";
      O     "Help_T107";
      O;
      AN    "COM_SHUTTLE".IN.Wozek_Auto_Info;
      A     "Na_Pozycji_KB1";
      A     "Marka_Jazdy_Na_Nowa_Poz";
      A     "Bezpieczne_Pokrycie_Foto";
      );
      R     "Zasprzeglenie_KB1";
NETWORK
TITLE =
NETWORK
TITLE = Wozek zasprzeglony do KB2
//Zasprzeglenie wozka w trybie recznym .Polaczone z funkcja FB8 
////KB2
      A     "Na_Pozycji_KB2";
      =     L 0.0;
      A     L 0.0;
      A     "KB2_Auto_Reczny";
      A     "Przejmij_Z_KB2";
      AN    "Marka_Jazdy_Na_Nowa_Poz";
      S     "Zasprzeglenie_KB2";
      A     L 0.0;
      A(;
      AN    "KB2_Auto_Reczny";
      A     "KB2_PB_Semi_Auto";
      O     "KB2_Przej_Auto_Na_Recz";
      O     "Warunk_Zasprz_KB2";
      );
      AN    "Marka_Jazdy_Na_Nowa_Poz";
      S     "Wozek_Na_Reczny";
      R     "Wozek_Na_Auto";
      S     "Zasprzeglenie_KB2";
      R     "Marka_Jazdy_Na_Nowa_Poz";
      A(;
      A     L 0.0;
      A     "KB2_Auto_Reczny";
      A     "KB2_PB_Auto";
      L     S5T#1S;
      SD    "Timer_103_KB2";
      NOP   0;
      NOP   0;
      NOP   0;
      A     "Timer_103_KB2";
      );
      AN    "Marka_Jazdy_Na_Nowa_Poz";
      =     L 0.1;
      A     L 0.1;
      BLD   102;
      S     "Wozek_Na_Auto";
      A     L 0.1;
      BLD   102;
      R     "Wozek_Na_Reczny";
      A     L 0.1;
      AN    "DB_CONECTOR_KB2".Winda.Foto_2;
      AN    "Foto_Pokryte_Czasowo";
      R     "Zasprzeglenie_KB2";
NETWORK
TITLE = Wozek zasprzeglony do KB2
//Przejmij kod kolbusa 2
////KB2
      A     "Zasprzeglenie_KB2";
      A(;
      A     "KB2_Auto_Reczny";
      A     "Na_Pozycji_KB2";
      A     "Foto_Wozek_Przod";
      A     "Foto_Wozek_Tyl";
      A     "Foto_Pokryte_Czasowo";
      O     "Help_T107";
      O;
      AN    "COM_SHUTTLE".IN.Wozek_Auto_Info;
      A     "Na_Pozycji_KB2";
      A     "Marka_Jazdy_Na_Nowa_Poz";
      A     "Bezpieczne_Pokrycie_Foto";
      );
      R     "Zasprzeglenie_KB2";
NETWORK
TITLE =
NETWORK
TITLE = Zasprzeglenie Intro pobieranie
//Zasprzeglenie wozka w trybie recznym .Polaczone z funkcja FB8 
////pobieranie I1
      A     "Na_Pozycji_Pob_I1";
      =     L 0.0;
      A     L 0.0;
      A     "I1_Buf_Auto_Reczny";
      A     "Przejmij_Z_I1";
      AN    "Marka_Jazdy_Na_Nowa_Poz";
      S     "Zasprzeglenie_Pob_I1";
      A     L 0.0;
      A(;
      AN    "I1_Buf_Auto_Reczny";
      A     "Buff_PB_Semi_Auto";
      O     "Buff_Przejscie_Na_Recz";
      O     "Warunk_Zasprz_Buffory";
      );
      AN    "Marka_Jazdy_Na_Nowa_Poz";
      S     "Wozek_Na_Reczny";
      R     "Wozek_Na_Auto";
      S     "Zasprzeglenie_Pob_I1";
      R     "Marka_Jazdy_Na_Nowa_Poz";
      A(;
      A     L 0.0;
      A     "I1_Buf_Auto_Reczny";
      A     "Buff_PB_Auto";
      L     S5T#1S;
      SD    "Timmer_104_Pobieranie";
      NOP   0;
      NOP   0;
      NOP   0;
      A     "Timmer_104_Pobieranie";
      );
      AN    "Marka_Jazdy_Na_Nowa_Poz";
      =     L 0.1;
      A     L 0.1;
      BLD   102;
      S     "Wozek_Na_Auto";
      A     L 0.1;
      BLD   102;
      R     "Wozek_Na_Reczny";
      A     L 0.1;
      AN    "DB_CONNECTOR_BUFF".Banda_16.Foto_1;
      AN    "Foto_Pokryte_Czasowo";
      R     "Zasprzeglenie_Pob_I1";
NETWORK
TITLE = Zasprzeglenie Intro pobieranie
////I1 pobieranie
      A     "Zasprzeglenie_Pob_I1";
      A(;
      A     "I1_Buf_Auto_Reczny";
      A     "Na_Pozycji_Pob_I1";
      A     "Foto_Wozek_Przod";
      A     "Foto_Wozek_Tyl";
      A     "Foto_Pokryte_Czasowo";
      O     "Help_T107";
      O;
      AN    "COM_SHUTTLE".IN.Wozek_Auto_Info;
      A     "Na_Pozycji_Pob_I1";
      A     "Marka_Jazdy_Na_Nowa_Poz";
      A     "Bezpieczne_Pokrycie_Foto";
      );
      R     "Zasprzeglenie_Pob_I1";
NETWORK
TITLE =
NETWORK
TITLE = Zasprzeglenie Intro pobieranie
//Zasprzeglenie wozka w trybie recznym .Polaczone z funkcja FB8 
////pobieranie I2
      A     "Na_Pozycji_Pob_I2";
      =     L 0.0;
      A     L 0.0;
      A     "I2_I3_Buf_Auto_Reczny";
      A     "Przejmij_z_I2";
      AN    "Marka_Jazdy_Na_Nowa_Poz";
      S     "Zasprzeglenie_Pob_I2";
      A     L 0.0;
      A(;
      AN    "I2_I3_Buf_Auto_Reczny";
      A     "Buff_2_PB_Semi_Auto";
      O     "Buff_Przejscie_Na_Recz";
      O     "Warunk_Zasprz_Buffory";
      );
      AN    "Marka_Jazdy_Na_Nowa_Poz";
      S     "Wozek_Na_Reczny";
      R     "Wozek_Na_Auto";
      S     "Zasprzeglenie_Pob_I2";
      R     "Marka_Jazdy_Na_Nowa_Poz";
      A(;
      A     L 0.0;
      A     "I2_I3_Buf_Auto_Reczny";
      A     "Buff_2_PB_Auto";
      L     S5T#1S;
      SD    "Timmer_Pob_I2";
      NOP   0;
      NOP   0;
      NOP   0;
      A     "Timmer_Pob_I2";
      );
      AN    "Marka_Jazdy_Na_Nowa_Poz";
      =     L 0.1;
      A     L 0.1;
      BLD   102;
      S     "Wozek_Na_Auto";
      A     L 0.1;
      BLD   102;
      R     "Wozek_Na_Reczny";
      A     L 0.1;
      AN    "DB_CONNECTOR_BUFF".Banda_8.Foto_1;
      AN    "Foto_Pokryte_Czasowo";
      R     "Zasprzeglenie_Pob_I2";
NETWORK
TITLE = Zasprzeglenie Intro pobieranie
////I2 pobieranie
      A     "Zasprzeglenie_Pob_I2";
      A(;
      A     "I2_I3_Buf_Auto_Reczny";
      A     "Na_Pozycji_Pob_I2";
      A     "Foto_Wozek_Przod";
      A     "Foto_Wozek_Tyl";
      A     "Foto_Pokryte_Czasowo";
      O     "Help_T107";
      O;
      AN    "COM_SHUTTLE".IN.Wozek_Auto_Info;
      A     "Na_Pozycji_Pob_I2";
      A     "Marka_Jazdy_Na_Nowa_Poz";
      A     "Bezpieczne_Pokrycie_Foto";
      );
      R     "Zasprzeglenie_Pob_I2";
NETWORK
TITLE =
NETWORK
TITLE = Zasprzeglenie Intro pobieranie
//Zasprzeglenie wozka w trybie recznym .Polaczone z funkcja FB8 
////pobieranie I3
      A     "Na_Pozycji_Pob_I3";
      =     L 0.0;
      A     L 0.0;
      A     "I2_I3_Buf_Auto_Reczny";
      A     "Przejmij_z_I3";
      AN    "Marka_Jazdy_Na_Nowa_Poz";
      S     "Zasprzeglenie_Pob_I3";
      A     L 0.0;
      A(;
      AN    "I2_I3_Buf_Auto_Reczny";
      A     "Buff_2_PB_Semi_Auto";
      O     "Buff_Przejscie_Na_Recz";
      O     "Warunk_Zasprz_Buffory";
      );
      AN    "Marka_Jazdy_Na_Nowa_Poz";
      S     "Wozek_Na_Reczny";
      R     "Wozek_Na_Auto";
      S     "Zasprzeglenie_Pob_I3";
      R     "Marka_Jazdy_Na_Nowa_Poz";
      A(;
      A     L 0.0;
      A     "I2_I3_Buf_Auto_Reczny";
      A     "Buff_2_PB_Auto";
      L     S5T#1S;
      SD    "Timmer_Pob_I3";
      NOP   0;
      NOP   0;
      NOP   0;
      A     "Timmer_Pob_I3";
      );
      AN    "Marka_Jazdy_Na_Nowa_Poz";
      =     L 0.1;
      A     L 0.1;
      BLD   102;
      S     "Wozek_Na_Auto";
      A     L 0.1;
      BLD   102;
      R     "Wozek_Na_Reczny";
      A     L 0.1;
      AN    "DB_CONNECTOR_BUFF".Banda_18.Foto_1;
      AN    "Foto_Pokryte_Czasowo";
      R     "Zasprzeglenie_Pob_I3";
NETWORK
TITLE = Zasprzeglenie Intro pobieranie
////I3 pobieranie
      A     "Zasprzeglenie_Pob_I3";
      A(;
      A     "I2_I3_Buf_Auto_Reczny";
      A     "Na_Pozycji_Pob_I3";
      A     "Foto_Wozek_Przod";
      A     "Foto_Wozek_Tyl";
      A     "Foto_Pokryte_Czasowo";
      O     "Help_T107";
      O;
      AN    "COM_SHUTTLE".IN.Wozek_Auto_Info;
      A     "Na_Pozycji_Pob_I3";
      A     "Marka_Jazdy_Na_Nowa_Poz";
      A     "Bezpieczne_Pokrycie_Foto";
      );
      R     "Zasprzeglenie_Pob_I3";
NETWORK
TITLE =
NETWORK
TITLE = Wozek zasprzeglony do Gender
////gender
      A     "Na_Pozycji_Gender";
      =     L 0.0;
      A     L 0.0;
      A     "Oddaj_Na_Spedycje";
      AN    "Marka_Jazdy_Na_Nowa_Poz";
      S     "Zasprzeglenie_Gender";
      A     L 0.0;
      A(;
      AN    "Gender_Auto_Reczny";
      A     "COM_GENDER".IN.PB_Reczny;
      O     "Gen_Przejscie_Na_Reczny";
      O     "Warunk_Zasprz_Gender";
      );
      AN    "Marka_Jazdy_Na_Nowa_Poz";
      S     "Wozek_Na_Reczny";
      R     "Wozek_Na_Auto";
      S     "Zasprzeglenie_Gender";
      R     "Marka_Jazdy_Na_Nowa_Poz";
      A(;
      A     L 0.0;
      A     "Gender_Auto_Reczny";
      A     "COM_GENDER".IN.PB_Auto;
      L     S5T#1S;
      SD    "T_100_Wozek_Na_Auto";
      NOP   0;
      NOP   0;
      NOP   0;
      A     "T_100_Wozek_Na_Auto";
      );
      AN    "Marka_Jazdy_Na_Nowa_Poz";
      AN    "DB_HMI_Wozek".HMI_IN.Wozek_W_Trybie_Auto;
      S     "Wozek_Na_Auto";
      R     "Wozek_Na_Reczny";
NETWORK
TITLE = Wozek zasprzeglony do Gender
////Gender
//
      A     "Zasprzeglenie_Gender";
      A(;
      A     "Gender_Auto_Reczny";
      A     "Na_Pozycji_Gender";
      AN    "Foto_Wozek_Przod";
      AN    "Foto_Wozek_Tyl";
      A     "Foto_Odkryte_Czasowo";
      O     "Help_T107";
      O;
      AN    "COM_SHUTTLE".IN.Wozek_Auto_Info;
      A     "Na_Pozycji_Gender";
      A     "Marka_Jazdy_Na_Nowa_Poz";
      A     "Bezpieczne_Pokrycie_Foto";
      );
      R     "Zasprzeglenie_Gender";
NETWORK
TITLE =
NETWORK
TITLE = Wozek zasprzeglony do odbierania
////odbieranie
      A     "Na_Pozycji_Odbieranie";
      =     L 0.0;
      A     L 0.0;
      A     "Oddaj_Na_Intro";
      AN    "Marka_Jazdy_Na_Nowa_Poz";
      S     "Zasprzeglenie_Odbieranie";
      A     L 0.0;
      A(;
      AN    "I1_Buf_Auto_Reczny";
      A     "Buff_PB_Semi_Auto";
      O     "Buff_Przejscie_Na_Recz";
      O     "Warunk_Zasprz_Buffory";
      );
      AN    "Marka_Jazdy_Na_Nowa_Poz";
      S     "Wozek_Na_Reczny";
      R     "Wozek_Na_Auto";
      S     "Zasprzeglenie_Odbieranie";
      R     "Marka_Jazdy_Na_Nowa_Poz";
      A(;
      A     L 0.0;
      A     "I1_Buf_Auto_Reczny";
      A     "Buff_PB_Auto";
      L     S5T#1S;
      SD    "Timmer_105_Odbieranie";
      NOP   0;
      NOP   0;
      NOP   0;
      A     "Timmer_105_Odbieranie";
      );
      AN    "Marka_Jazdy_Na_Nowa_Poz";
      S     "Wozek_Na_Auto";
      R     "Wozek_Na_Reczny";
NETWORK
TITLE = Wozek zasprzeglony do odbierania
////odbieranie
//
      A     "Zasprzeglenie_Odbieranie";
      A(;
      A     "I1_Buf_Auto_Reczny";
      A     "Na_Pozycji_Odbieranie";
      AN    "Foto_Wozek_Przod";
      AN    "Foto_Wozek_Tyl";
      A     "Foto_Odkryte_Czasowo";
      O     "Help_T107";
      O;
      AN    "COM_SHUTTLE".IN.Wozek_Auto_Info;
      A     "Na_Pozycji_Odbieranie";
      A     "Marka_Jazdy_Na_Nowa_Poz";
      A     "Bezpieczne_Pokrycie_Foto";
      );
      R     "Zasprzeglenie_Odbieranie";
NETWORK
TITLE =
//Zasprzeglenie wozka
//
      A     "Zawsze_True";
      A(;
      O     "Zasprzeglenie_KB1";
      O     "Zasprzeglenie_KB2";
      O     "Zasprzeglenie_Gender";
      O     "Zasprzeglenie_Odbieranie";
      O     "Zasprzeglenie_Pob_I1";
      O     "Zasprzeglenie_Pob_I2";
      O     "Zasprzeglenie_Pob_I3";
      );
      R     "Rozprzeglenie_Wozka";
      S     "Zasprzegnij_Wozek";
NETWORK
TITLE =
//Rozprzeglenie wozka
//
      AN    "Zasprzeglenie_KB1";
      AN    "Zasprzeglenie_KB2";
      AN    "Zasprzeglenie_Gender";
      AN    "Zasprzeglenie_Odbieranie";
      AN    "Zasprzeglenie_Pob_I1";
      AN    "Zasprzeglenie_Pob_I2";
      AN    "Zasprzeglenie_Pob_I3";
      =     L 0.0;
      A     L 0.0;
      BLD   102;
      S     "Rozprzeglenie_Wozka";
      A     L 0.0;
      L     S5T#2S;
      SD    "T71_Opoznienie_Rozp";
      NOP   0;
      NOP   0;
      NOP   0;
      A     "T71_Opoznienie_Rozp";
      R     "Zasprzegnij_Wozek";
NETWORK
TITLE = Wozek zasprzeglony do odbierania
//Reset zasprzeglenia gdy to niemozliwe
      A     "Zawsze_True";
      =     L 0.0;
      A     L 0.0;
      AN    "Na_Pozycji_KB1";
      R     "Zasprzeglenie_KB1";
      A     L 0.0;
      AN    "Na_Pozycji_KB2";
      R     "Zasprzeglenie_KB2";
      A     L 0.0;
      AN    "Na_Pozycji_Gender";
      R     "Zasprzeglenie_Gender";
      A     L 0.0;
      AN    "Na_Pozycji_Odbieranie";
      R     "Zasprzeglenie_Odbieranie";
      A     L 0.0;
      AN    "Na_Pozycji_Pob_I1";
      R     "Zasprzeglenie_Pob_I1";
      A     L 0.0;
      AN    "Na_Pozycji_Pob_I2";
      R     "Zasprzeglenie_Pob_I2";
      A     L 0.0;
      AN    "Na_Pozycji_Pob_I3";
      R     "Zasprzeglenie_Pob_I3";
      A     L 0.0;
      AN    "Na_Pozycji_KB1";
      AN    "Na_Pozycji_KB2";
      AN    "Na_Pozycji_Gender";
      AN    "Na_Pozycji_Odbieranie";
      AN    "Na_Pozycji_Pob_I1";
      AN    "Na_Pozycji_Pob_I2";
      AN    "Na_Pozycji_Pob_I3";
      R     "Zasprzegnij_Wozek";
      S     "Rozprzeglenie_Wozka";
      R     "Wozek_Na_Reczny";
      R     "Wozek_Na_Auto";
NETWORK
TITLE =
      A(;
      AN    "Foto_Wozek_Przod";
      AN    "Foto_Wozek_Tyl";
      AN    "Brak_Komunikacji_Shuttle";
      L     S5T#3S;
      SD    "Help_T90";
      NOP   0;
      NOP   0;
      NOP   0;
      A     "Help_T90";
      );
      A(;
      L     "DB_HMI_Wozek".HMI_IN_OUT.Wartosc_Buforu_Wozek;
      L     L#0;
      <>D;
      );
      JNB   _001;
      L     L#0;
      T     "DB_HMI_Wozek".HMI_IN_OUT.Wartosc_Buforu_Wozek;
_001: NOP   0;
NETWORK
TITLE =
//Sprawdzenie czy wozek nie ma palety widmo jak ma to oddaje na buffory odbioru
      A     "Foto_Wozek_Przod";
      =     L 0.0;
      BLD   103;
      A     "Foto_Wozek_Tyl";
      =     L 0.1;
      BLD   103;
      A     "Zawsze_False";
      JNB   _002;
      CALL  "Monitor_Palety" (
           Foto_Pozycji_Przod       := L 0.0,
           Foto_Pozycji_Tyl         := L 0.1,
           iod_Wartosc_Rejestru     := "DB_HMI_Wozek".HMI_IN_OUT.Wartosc_Buforu_Wozek);
_002: NOP   0;
NETWORK
TITLE =
      A     "Foto_Wozek_Przod";
      A     "Foto_Wozek_Tyl";
      A     "Wozek_Auto_Reczny";
      L     S5T#2S;
      SD    "Timer_T1";
      NOP   0;
      NOP   0;
      NOP   0;
      A     "Timer_T1";
      =     "Help_Widmo";
NETWORK
TITLE =
      A     "Help_Widmo";
      =     L 0.0;
      BLD   103;
      CALL  "Znajdz_Widmo" (
           Paleta_Obecna            := L 0.0,
           iod_Wartosc_Rejestru     := "DB_HMI_Wozek".HMI_IN_OUT.Wartosc_Buforu_Wozek);
      NOP   0;
END_FUNCTION

FUNCTION "Sprawdzenie_Okna" : VOID	// FC 7
VERSION : 0.1
VAR_INPUT
  War_Pozycji_Aktualnej : DINT ;	//Pozycja aktualna w mm
  War_Pozycji_Zadanej : DINT ;
  War_Pozycji_Maszyn : DINT ;	//Pozycja zadana w mm
  Tolerancja : DINT ;	//Tolerancja w mm
END_VAR
VAR_OUTPUT
  Na_Pozycji_Maszyny : BOOL ;
  Na_Pozycji_Zadanej : BOOL ;
  Na_Poz_Zad_Masz : BOOL ;
END_VAR
VAR_TEMP
  Schowek_War_Gora : DINT ;
  Schowek_War_Dol : DINT ;
END_VAR
BEGIN
NETWORK
TITLE =
//Ten network celow jest wolny
NETWORK
TITLE =
//Gorny zakres
      L     #War_Pozycji_Maszyn;
      L     #Tolerancja;
      +D;
      T     #Schowek_War_Gora;
//Dolny zakres
      L     #War_Pozycji_Maszyn;
      L     #Tolerancja;
      -D;
      T     #Schowek_War_Dol;
//sprawdzenie
      L     #War_Pozycji_Aktualnej;
      L     #Schowek_War_Gora;
      <D;
      =     L 8.0;
      L     #War_Pozycji_Aktualnej;
      L     #Schowek_War_Dol;
      >D;
      =     L 8.1;
      A     L 8.1;
      A     L 8.0;
      =     L 9.0;
      =     #Na_Pozycji_Maszyny;
//Na pozycji zadanej   i pozycji maszyny
//Gorny zakres
      L     #War_Pozycji_Zadanej;
      L     #Tolerancja;
      +D;
      T     #Schowek_War_Gora;
//Dolny zakres
      L     #War_Pozycji_Zadanej;
      L     #Tolerancja;
      -D;
      T     #Schowek_War_Dol;
//sprawdzenie
      L     #War_Pozycji_Aktualnej;
      L     #Schowek_War_Gora;
      <D;
      =     L 8.2;
      L     #War_Pozycji_Aktualnej;
      L     #Schowek_War_Dol;
      >D;
      =     L 8.3;
      A     L 8.2;
      A     L 8.3;
      =     L 9.1;
      =     #Na_Pozycji_Zadanej;
//Na pozycji zadanej maszyny
      A     L 9.0;
      A     L 9.1;
      =     #Na_Poz_Zad_Masz;
END_FUNCTION

FUNCTION "Lenze_Sew_Shell_KB1" : VOID	// FC 8
AUTHOR : Kng
NAME : DRIVE
VERSION : 0.1
VAR_INPUT
  ESTOP : BOOL ;
  ADD_Falownika : INT ;
  Tryb : BOOL ;	//0-banda, tryb owijania
  Jazda_Lewo : BOOL ;
  Jazda_Prawo : BOOL ;
  Wolno : BOOL ;	//0-szybko,1-wolno
  V_Zadana : REAL ;	//Predkosc zadana w trybie owijania
END_VAR
VAR_OUTPUT
  Falownik_Gotowy : BOOL ;
  Odblokuj_Falownik : BOOL ;
  Odblokuj_Hamulec : BOOL ;
END_VAR
VAR_TEMP
  L_Blad_Falownika : BOOL ;
  L_Status_Word : WORD ;
  L_V_Zwracane : REAL ;
  L_Predkosc_Przejsciowa : REAL ;
  Temp_Bit_1 : BOOL ;
END_VAR
BEGIN
NETWORK
TITLE =
//Ten network celowo jest wolny
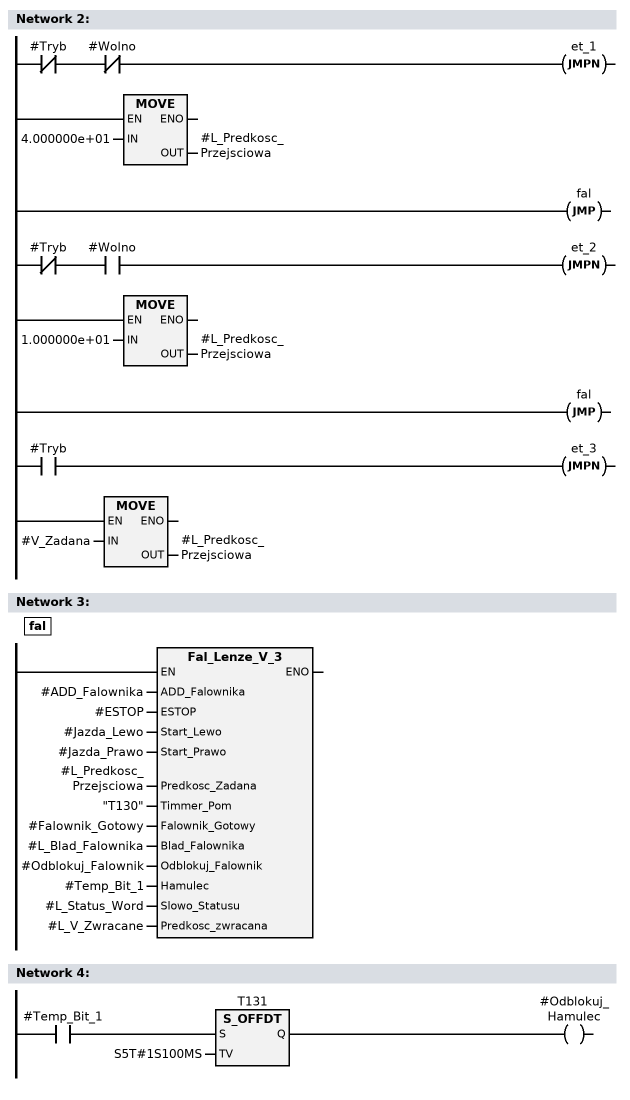
NETWORK
TITLE =
      AN    #Tryb;
      AN    #Wolno;
      JCN   et_1;
      L     4.000000e+01;
      T     #L_Predkosc_Przejsciowa;
      JU    fal;
et_1: NOP   0;
      AN    #Tryb;
      A     #Wolno;
      JCN   et_2;
      L     1.000000e+01;
      T     #L_Predkosc_Przejsciowa;
      JU    fal;
et_2: NOP   0;
      A     #Tryb;
      JCN   et_3;
      L     #V_Zadana;
      T     #L_Predkosc_Przejsciowa;
et_3: NOP   0;
NETWORK
TITLE =
//Opis Falownika
fal:  NOP   0;
      CALL  "Fal_Lenze_V_3" (
           ADD_Falownika            := #ADD_Falownika,
           ESTOP                    := #ESTOP,
           Start_Lewo               := #Jazda_Lewo,
           Start_Prawo              := #Jazda_Prawo,
           Predkosc_Zadana          := #L_Predkosc_Przejsciowa,
           Timmer_Pom               := "T130",
           Falownik_Gotowy          := #Falownik_Gotowy,
           Blad_Falownika           := #L_Blad_Falownika,
           Odblokuj_Falownik        := #Odblokuj_Falownik,
           Hamulec                  := #Temp_Bit_1,
           Slowo_Statusu            := #L_Status_Word,
           Predkosc_zwracana        := #L_V_Zwracane);
NETWORK
TITLE =
      A     #Temp_Bit_1;
      L     S5T#1S100MS;
      SF    "T131";
      NOP   0;
      NOP   0;
      NOP   0;
      A     "T131";
      =     #Odblokuj_Hamulec;
END_FUNCTION

FUNCTION "Lenze_Sew_Shell_KB2" : VOID	// FC 9
AUTHOR : Kng
NAME : DRIVE
VERSION : 0.1
VAR_INPUT
  ESTOP : BOOL ;
  ADD_Falownika : INT ;
  Tryb : BOOL ;	//0-banda, tryb owijania
  Jazda_Lewo : BOOL ;
  Jazda_Prawo : BOOL ;
  Wolno : BOOL ;	//0-szybko,1-wolno
  V_Zadana : REAL ;	//Predkosc zadana w trybie owijania
END_VAR
VAR_OUTPUT
  Falownik_Gotowy : BOOL ;
  Odblokuj_Falownik : BOOL ;
  Odblokuj_Hamulec : BOOL ;
END_VAR
VAR_TEMP
  L_Blad_Falownika : BOOL ;
  L_Status_Word : WORD ;
  L_V_Zwracane : REAL ;
  L_Predkosc_Przejsciowa : REAL ;
  Temp_Bit_1 : BOOL ;
END_VAR
BEGIN
NETWORK
TITLE =
//Ten network celowo jest wolny
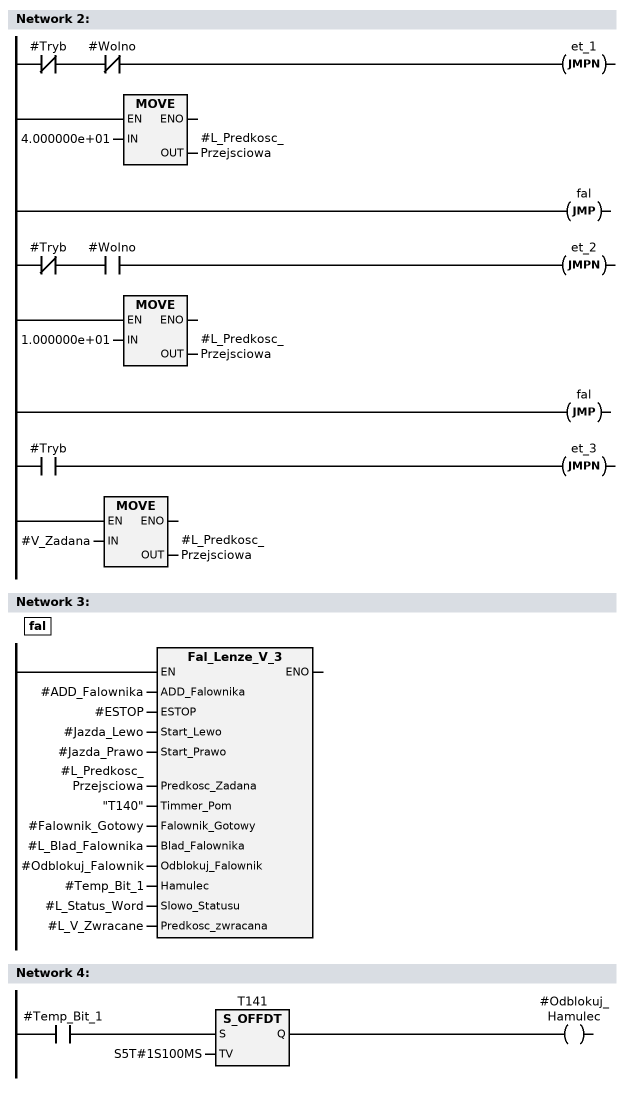
NETWORK
TITLE =
      AN    #Tryb;
      AN    #Wolno;
      JCN   et_1;
      L     4.000000e+01;
      T     #L_Predkosc_Przejsciowa;
      JU    fal;
et_1: NOP   0;
      AN    #Tryb;
      A     #Wolno;
      JCN   et_2;
      L     1.000000e+01;
      T     #L_Predkosc_Przejsciowa;
      JU    fal;
et_2: NOP   0;
      A     #Tryb;
      JCN   et_3;
      L     #V_Zadana;
      T     #L_Predkosc_Przejsciowa;
et_3: NOP   0;
NETWORK
TITLE =
//Opis Falownika
fal:  NOP   0;
      CALL  "Fal_Lenze_V_3" (
           ADD_Falownika            := #ADD_Falownika,
           ESTOP                    := #ESTOP,
           Start_Lewo               := #Jazda_Lewo,
           Start_Prawo              := #Jazda_Prawo,
           Predkosc_Zadana          := #L_Predkosc_Przejsciowa,
           Timmer_Pom               := "T140",
           Falownik_Gotowy          := #Falownik_Gotowy,
           Blad_Falownika           := #L_Blad_Falownika,
           Odblokuj_Falownik        := #Odblokuj_Falownik,
           Hamulec                  := #Temp_Bit_1,
           Slowo_Statusu            := #L_Status_Word,
           Predkosc_zwracana        := #L_V_Zwracane);
NETWORK
TITLE =
      A     #Temp_Bit_1;
      L     S5T#1S100MS;
      SF    "T141";
      NOP   0;
      NOP   0;
      NOP   0;
      A     "T141";
      =     #Odblokuj_Hamulec;
END_FUNCTION

FUNCTION "Fal_Lenze_V_3" : VOID	// FC 10
//Funkcja kontrolujaca Falownik Lenze.Zakladane jest ze obszar wejsc falownika 
//pokrywa sie z obszarem wyjsc(PIWX,PQWY,X=Y patrz Hardware).
//
//***CTW***
//POW1-S³owo  kontrolne 1 (CTW)
//POW2-Predkosc zadana (NSET1-N1):+-480HZ=+-24000
//**STW***
//PIW1-S³owo statusu 1 (STW)
//PIW2-Czestotliwosc wyjsciowa+poslizg
//
//
//-Wyroznia sie nastepujace s³owa sterujace:
//CTW:0000 0000 0111 1110 (007E)-falownik gotowy do startu/Funkcja Stop
//CTW:0000 0000 0111 1111 (007F)-falownik zostaje uruchominony
//CTW:xxxx xxxx xxxx x01x (x-wszystko jedno)-falownik zatrzymany Szybki Stop
//-Wyroznia sie nastepujace s³owa statusu:
//STW:xxxx xxxx x01x 0001-Falownik gotowy do startu
//STW:xxxx xxxx x01x 0111-Falownik pracuje
//STW:xxxx xxxx x0xx 1000-Blad Falownika 
//
//
//
AUTHOR : Kng
NAME : DRIVE
VERSION : 0.1
VAR_INPUT
  ADD_Falownika : INT ;
  ESTOP : BOOL ;	//Szybki Stop Falownika
  Start_Lewo : BOOL ;	//Start Falownika CW
  Start_Prawo : BOOL ;	//Start Falownika CCW
  Predkosc_Zadana : REAL ;	//Predkosc silnika w Hz
  Timmer_Pom : TIMER ;	//Timmer pomocniczy
END_VAR
VAR_OUTPUT
  Falownik_Gotowy : BOOL ;
  Blad_Falownika : BOOL ;	//Falownik zwraca blad
  Odblokuj_Falownik : BOOL ;	//Przekaznik_Odblokowujacy
  Hamulec : BOOL ;	//Odblokowanie hamulca
  Slowo_Statusu : WORD ;	//Slowo Satusu falownika
  Predkosc_zwracana : REAL ;	//Predkosc zwracana przez Falownik
END_VAR
VAR_TEMP
  Adres_1 : DWORD ;
  Adres_2 : DWORD ;
  STW : WORD ;
  CTW : BOOL ;
  H_Temp : INT ;
  H_Temp_2 : INT ;
  Help_Bool_1 : BOOL ;
  Adres_3 : DWORD ;
  Timmer_Name : WORD ;
END_VAR
BEGIN
NETWORK
TITLE =
//Wskaznik do falownika
//********************************Wyliczenie Adresow
      L     #ADD_Falownika;
      SLD   3;
      T     #Adres_1;	//adres falownika control word
      L     #ADD_Falownika;
      L     2;
      +I;
      SLD   3;
      T     #Adres_2;	//adres falownika predkosc
      L     PIW [#Adres_1];	//zaladuj stw
      T     #STW;	//Slowo statusu
      T     #Slowo_Statusu;	//LW8
NETWORK
TITLE =
//Tworzenie slowa kontrolnego
// (network holds code this reader does not know; not shown)
//*********************************Blad Falownika
//*********************************Falownik gotowy do pracy
//**********************************Odblokuj falownik
//*********************************E-Stop Falownika
//*********************************Stop Falownika
//*********************************Start Falownika
//**
//      A     "Zawsze_False"
//*********************************Zaden z powyzszych warunkow
NETWORK
TITLE =
//Odczyt predkosc z falownika oraz  przypisanie predkosci od falownika.
//Zakres prekosci falownika:
//+-480HZ=+-24000
//
//1Hz=50 jednostek(dokladnosc 0.1Hz+pó³ cyfry)
//Predkosc bedzie zaokraglona do jednego miejsca po przecinku
//
//Predkosc zadana (zaokraglona z real do int)
//********************************Zadanie predkosci
pre1: L     #Predkosc_Zadana;	//50
      L     2.000000e+00;	//2
      /R;	//25
      L     1.000000e+02;
      *R;
      A     #Start_Prawo;
      JCN   e1;
      L     -1.000000e+00;
      *R;
e1:   RND;
pre2: T     #H_Temp;
      L     #H_Temp;
      T     PQW [#Adres_2];	//Transfer predkosci
//********************************Odczyt predkosci
//********************************
      L     PIW [#Adres_2];
      ITD;
      DTR;
      L     2.000000e+00;
      *R;
      L     1.000000e+02;
      /R;
      T     #Predkosc_zwracana;
      L     0.000000e+00;	//predkosc odczytna z falownika
      ==R;
      R     #Hamulec;
END_FUNCTION

FUNCTION "Przyciski_Dwufunkcyjne" : VOID	// FC 11
AUTHOR : Kng
NAME : Help_FC
VERSION : 0.1
VAR_INPUT
  Kierunek_Prawo : BOOL ;
  Kierunek_Lewo : BOOL ;
  Funkcja : BOOL ;
END_VAR
VAR_OUTPUT
  Jazda_Prawo : BOOL ;
  Jazda_Lewo : BOOL ;
  Obrot_Prawo : BOOL ;
  Obrot_Lewo : BOOL ;
END_VAR
BEGIN
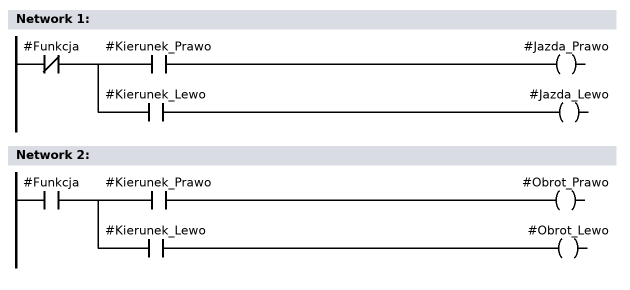
NETWORK
TITLE =
      AN    #Funkcja;
      =     L 0.0;
      A     L 0.0;
      A     #Kierunek_Prawo;
      =     #Jazda_Prawo;
      A     L 0.0;
      A     #Kierunek_Lewo;
      =     #Jazda_Lewo;
NETWORK
TITLE =
      A     #Funkcja;
      =     L 0.0;
      A     L 0.0;
      A     #Kierunek_Prawo;
      =     #Obrot_Prawo;
      A     L 0.0;
      A     #Kierunek_Lewo;
      =     #Obrot_Lewo;
END_FUNCTION

FUNCTION "Auto_Reczny_KB1" : VOID	// FC 13
AUTHOR : Kng
NAME : KB1
VERSION : 0.1
BEGIN
NETWORK
TITLE =
NETWORK
TITLE =
//Ten network celowo jest wolny
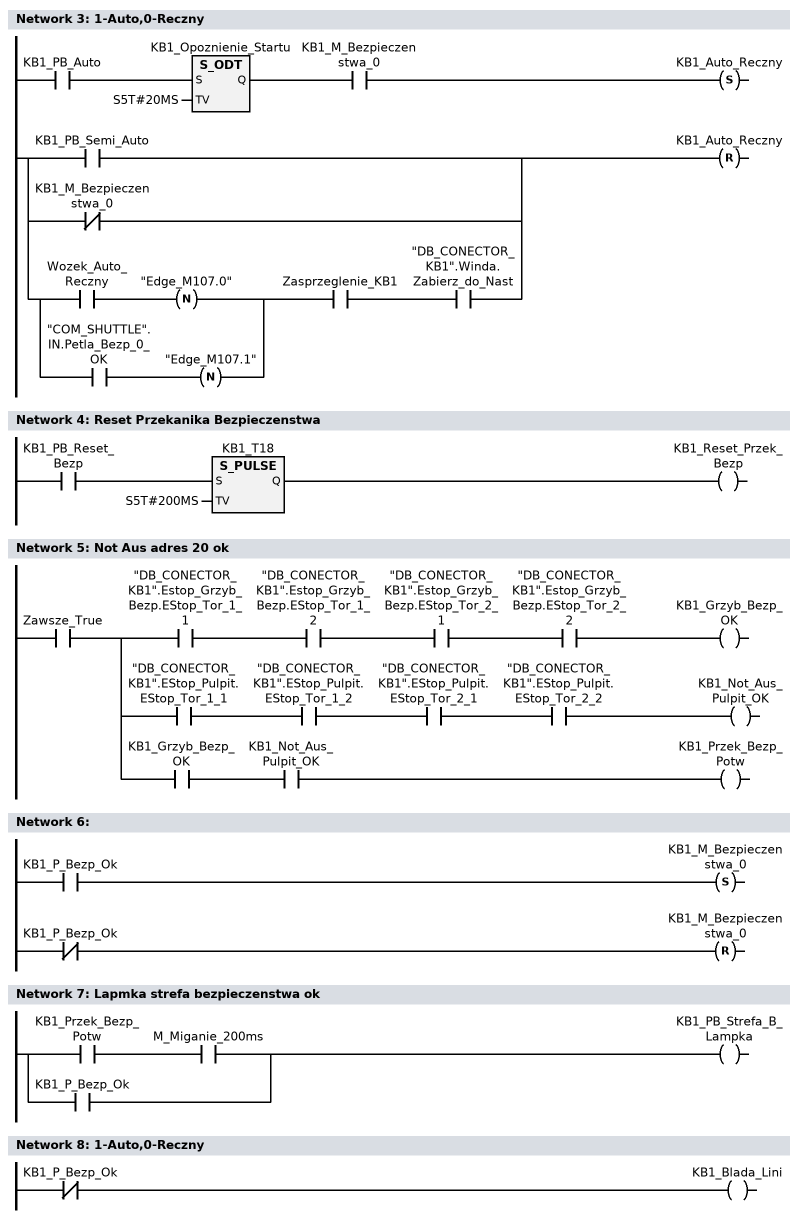
NETWORK
TITLE = 1-Auto,0-Reczny
//Wybranie trybu auto
      A(;
      A     "KB1_PB_Auto";
      L     S5T#20MS;
      SD    "KB1_Opoznienie_Startu";
      NOP   0;
      NOP   0;
      NOP   0;
      A     "KB1_Opoznienie_Startu";
      );
      A     "KB1_M_Bezpieczenstwa_0";
      S     "KB1_Auto_Reczny";
      A(;
      O     "KB1_PB_Semi_Auto";
      ON    "KB1_M_Bezpieczenstwa_0";
      O(;
      A(;
      A     "Wozek_Auto_Reczny";
      FN    "Edge_M107.0";
      O(;
      A     "COM_SHUTTLE".IN.Petla_Bezp_0_OK;
      FN    "Edge_M107.1";
      );
      );
      A     "Zasprzeglenie_KB1";
      A     "DB_CONECTOR_KB1".Winda.Zabierz_do_Nast;
      );
      );
      R     "KB1_Auto_Reczny";
      NOP   0;
NETWORK
TITLE = Reset Przekanika Bezpieczenstwa
//Reset przekanika bezpieczenstwa
//
      A     "KB1_PB_Reset_Bezp";
      L     S5T#200MS;
      SP    "KB1_T18";
      NOP   0;
      NOP   0;
      NOP   0;
      A     "KB1_T18";
      =     "KB1_Reset_Przek_Bezp";
NETWORK
TITLE = Not Aus adres 20 ok
//Sprawdzenie czy mozna potwierdzic przekaznik bezpieczenstwa
      A     "Zawsze_True";
      =     L 0.0;
      A     L 0.0;
      A     "DB_CONECTOR_KB1".Estop_Grzyb_Bezp.EStop_Tor_1_1;
      A     "DB_CONECTOR_KB1".Estop_Grzyb_Bezp.EStop_Tor_1_2;
      A     "DB_CONECTOR_KB1".Estop_Grzyb_Bezp.EStop_Tor_2_1;
      A     "DB_CONECTOR_KB1".Estop_Grzyb_Bezp.EStop_Tor_2_2;
      =     "KB1_Grzyb_Bezp_OK";
      A     L 0.0;
      A     "DB_CONECTOR_KB1".EStop_Pulpit.EStop_Tor_1_1;
      A     "DB_CONECTOR_KB1".EStop_Pulpit.EStop_Tor_1_2;
      A     "DB_CONECTOR_KB1".EStop_Pulpit.EStop_Tor_2_1;
      A     "DB_CONECTOR_KB1".EStop_Pulpit.EStop_Tor_2_2;
      =     "KB1_Not_Aus_Pulpit_OK";
      A     L 0.0;
      A     "KB1_Grzyb_Bezp_OK";
      A     "KB1_Not_Aus_Pulpit_OK";
      =     "KB1_Przek_Bezp_Potw";
NETWORK
TITLE =
      A     "KB1_P_Bezp_Ok";
      S     "KB1_M_Bezpieczenstwa_0";
      AN    "KB1_P_Bezp_Ok";
      R     "KB1_M_Bezpieczenstwa_0";
      NOP   0;
NETWORK
TITLE = Lapmka strefa bezpieczenstwa ok
      A     "KB1_Przek_Bezp_Potw";
      A     "M_Miganie_200ms";
      O     "KB1_P_Bezp_Ok";
      =     "KB1_PB_Strefa_B_Lampka";
NETWORK
TITLE = 1-Auto,0-Reczny
//Lampka wieza sygnalizacyjna
      AN    "KB1_P_Bezp_Ok";
      =     "KB1_Blada_Lini";
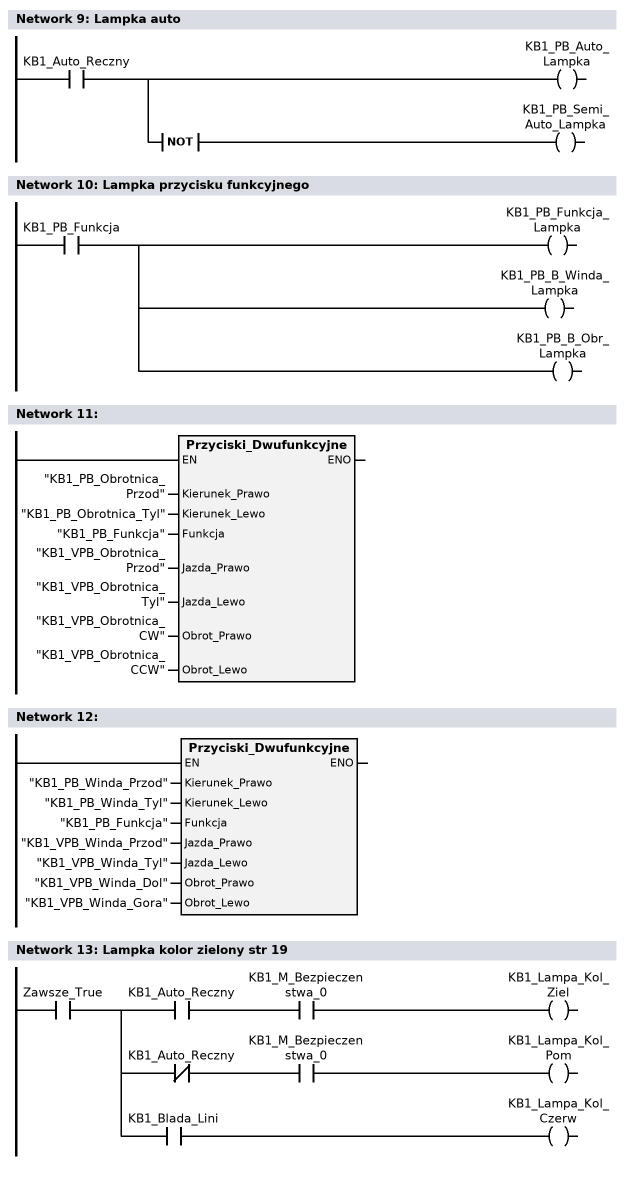
NETWORK
TITLE = Lampka auto
      A     "KB1_Auto_Reczny";
      =     L 0.0;
      A     L 0.0;
      BLD   102;
      =     "KB1_PB_Auto_Lampka";
      A     L 0.0;
      NOT;
      =     "KB1_PB_Semi_Auto_Lampka";
NETWORK
TITLE = Lampka przycisku funkcyjnego
//Lampka przycisk Funkcyjny
      A     "KB1_PB_Funkcja";
      =     "KB1_PB_Funkcja_Lampka";
      =     "KB1_PB_B_Winda_Lampka";
      =     "KB1_PB_B_Obr_Lampka";
NETWORK
TITLE =
//przycisk funkcyjny obrotnica
//
      CALL  "Przyciski_Dwufunkcyjne" (
           Kierunek_Prawo           := "KB1_PB_Obrotnica_Przod",
           Kierunek_Lewo            := "KB1_PB_Obrotnica_Tyl",
           Funkcja                  := "KB1_PB_Funkcja",
           Jazda_Prawo              := "KB1_VPB_Obrotnica_Przod",
           Jazda_Lewo               := "KB1_VPB_Obrotnica_Tyl",
           Obrot_Prawo              := "KB1_VPB_Obrotnica_CW",
           Obrot_Lewo               := "KB1_VPB_Obrotnica_CCW");
NETWORK
TITLE =
//przycisk funkcyjny winda
//
      CALL  "Przyciski_Dwufunkcyjne" (
           Kierunek_Prawo           := "KB1_PB_Winda_Przod",
           Kierunek_Lewo            := "KB1_PB_Winda_Tyl",
           Funkcja                  := "KB1_PB_Funkcja",
           Jazda_Prawo              := "KB1_VPB_Winda_Przod",
           Jazda_Lewo               := "KB1_VPB_Winda_Tyl",
           Obrot_Prawo              := "KB1_VPB_Winda_Dol",
           Obrot_Lewo               := "KB1_VPB_Winda_Gora");
NETWORK
TITLE = Lampka kolor zielony str 19
//Lampki wieza sygnalizacyjna
      A     "Zawsze_True";
      =     L 0.0;
      A     L 0.0;
      A     "KB1_Auto_Reczny";
      A     "KB1_M_Bezpieczenstwa_0";
      =     "KB1_Lampa_Kol_Ziel";
      A     L 0.0;
      AN    "KB1_Auto_Reczny";
      A     "KB1_M_Bezpieczenstwa_0";
      =     "KB1_Lampa_Kol_Pom";
      A     L 0.0;
      A     "KB1_Blada_Lini";
      =     "KB1_Lampa_Kol_Czerw";
END_FUNCTION

FUNCTION "Auto_Reczny_KB2" : VOID	// FC 14
AUTHOR : Kng
NAME : KB2
VERSION : 0.1
BEGIN
NETWORK
TITLE =
NETWORK
TITLE =
//Ten network celowo jest wolny
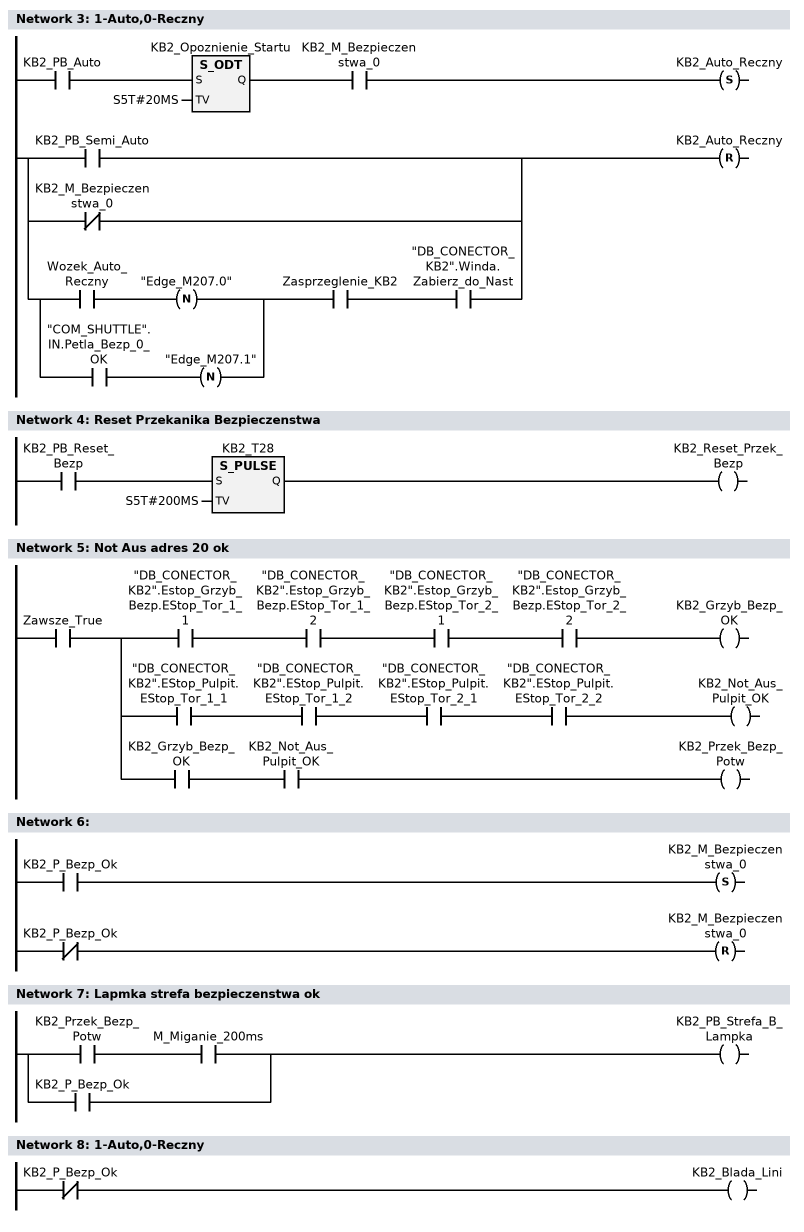
NETWORK
TITLE = 1-Auto,0-Reczny
//Wybranie trybu auto
      A(;
      A     "KB2_PB_Auto";
      L     S5T#20MS;
      SD    "KB2_Opoznienie_Startu";
      NOP   0;
      NOP   0;
      NOP   0;
      A     "KB2_Opoznienie_Startu";
      );
      A     "KB2_M_Bezpieczenstwa_0";
      S     "KB2_Auto_Reczny";
      A(;
      O     "KB2_PB_Semi_Auto";
      ON    "KB2_M_Bezpieczenstwa_0";
      O(;
      A(;
      A     "Wozek_Auto_Reczny";
      FN    "Edge_M207.0";
      O(;
      A     "COM_SHUTTLE".IN.Petla_Bezp_0_OK;
      FN    "Edge_M207.1";
      );
      );
      A     "Zasprzeglenie_KB2";
      A     "DB_CONECTOR_KB2".Winda.Zabierz_do_Nast;
      );
      );
      R     "KB2_Auto_Reczny";
      NOP   0;
NETWORK
TITLE = Reset Przekanika Bezpieczenstwa
//Reset przekanika bezpieczenstwa
//
      A     "KB2_PB_Reset_Bezp";
      L     S5T#200MS;
      SP    "KB2_T28";
      NOP   0;
      NOP   0;
      NOP   0;
      A     "KB2_T28";
      =     "KB2_Reset_Przek_Bezp";
NETWORK
TITLE = Not Aus adres 20 ok
//Sprawdzenie czy mozna potwierdzic przekaznik bezpieczenstwa
      A     "Zawsze_True";
      =     L 0.0;
      A     L 0.0;
      A     "DB_CONECTOR_KB2".Estop_Grzyb_Bezp.EStop_Tor_1_1;
      A     "DB_CONECTOR_KB2".Estop_Grzyb_Bezp.EStop_Tor_1_2;
      A     "DB_CONECTOR_KB2".Estop_Grzyb_Bezp.EStop_Tor_2_1;
      A     "DB_CONECTOR_KB2".Estop_Grzyb_Bezp.EStop_Tor_2_2;
      =     "KB2_Grzyb_Bezp_OK";
      A     L 0.0;
      A     "DB_CONECTOR_KB2".EStop_Pulpit.EStop_Tor_1_1;
      A     "DB_CONECTOR_KB2".EStop_Pulpit.EStop_Tor_1_2;
      A     "DB_CONECTOR_KB2".EStop_Pulpit.EStop_Tor_2_1;
      A     "DB_CONECTOR_KB2".EStop_Pulpit.EStop_Tor_2_2;
      =     "KB2_Not_Aus_Pulpit_OK";
      A     L 0.0;
      A     "KB2_Grzyb_Bezp_OK";
      A     "KB2_Not_Aus_Pulpit_OK";
      =     "KB2_Przek_Bezp_Potw";
NETWORK
TITLE =
      A     "KB2_P_Bezp_Ok";
      S     "KB2_M_Bezpieczenstwa_0";
      AN    "KB2_P_Bezp_Ok";
      R     "KB2_M_Bezpieczenstwa_0";
      NOP   0;
NETWORK
TITLE = Lapmka strefa bezpieczenstwa ok
      A     "KB2_Przek_Bezp_Potw";
      A     "M_Miganie_200ms";
      O     "KB2_P_Bezp_Ok";
      =     "KB2_PB_Strefa_B_Lampka";
NETWORK
TITLE = 1-Auto,0-Reczny
//Lampka wieza sygnalizacyjna
      AN    "KB2_P_Bezp_Ok";
      =     "KB2_Blada_Lini";
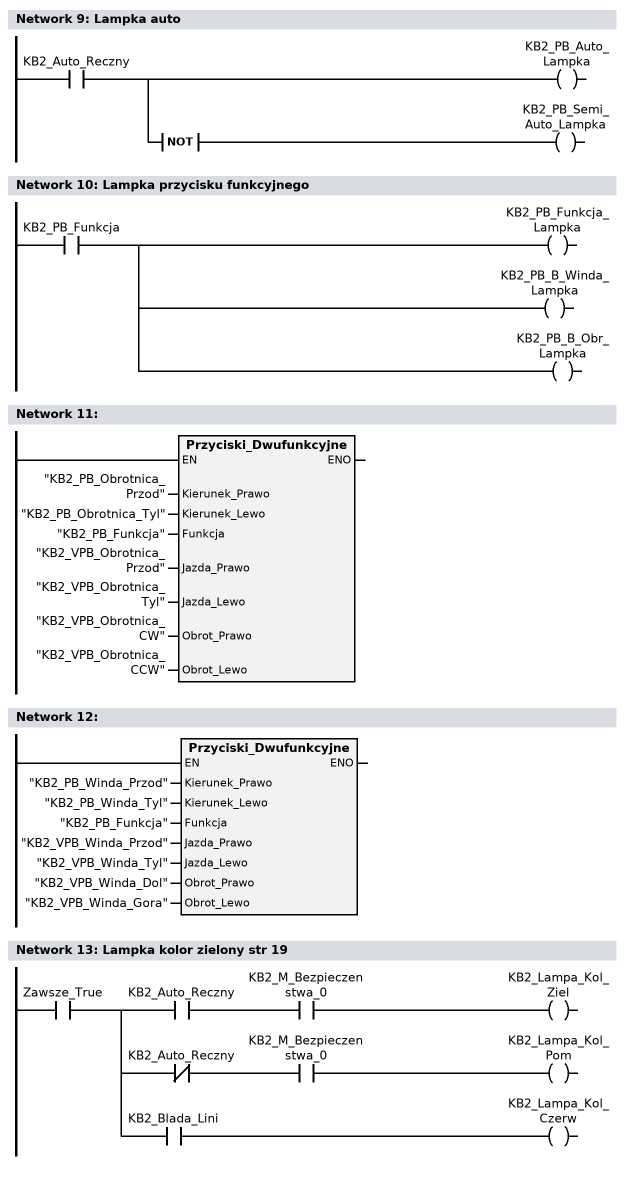
NETWORK
TITLE = Lampka auto
      A     "KB2_Auto_Reczny";
      =     L 0.0;
      A     L 0.0;
      BLD   102;
      =     "KB2_PB_Auto_Lampka";
      A     L 0.0;
      NOT;
      =     "KB2_PB_Semi_Auto_Lampka";
NETWORK
TITLE = Lampka przycisku funkcyjnego
//Lampka przycisk Funkcyjny
      A     "KB2_PB_Funkcja";
      =     "KB2_PB_Funkcja_Lampka";
      =     "KB2_PB_B_Winda_Lampka";
      =     "KB2_PB_B_Obr_Lampka";
NETWORK
TITLE =
//przycisk funkcyjny obrotnica
//
      CALL  "Przyciski_Dwufunkcyjne" (
           Kierunek_Prawo           := "KB2_PB_Obrotnica_Przod",
           Kierunek_Lewo            := "KB2_PB_Obrotnica_Tyl",
           Funkcja                  := "KB2_PB_Funkcja",
           Jazda_Prawo              := "KB2_VPB_Obrotnica_Przod",
           Jazda_Lewo               := "KB2_VPB_Obrotnica_Tyl",
           Obrot_Prawo              := "KB2_VPB_Obrotnica_CW",
           Obrot_Lewo               := "KB2_VPB_Obrotnica_CCW");
NETWORK
TITLE =
//przycisk funkcyjny winda
//
      CALL  "Przyciski_Dwufunkcyjne" (
           Kierunek_Prawo           := "KB2_PB_Winda_Przod",
           Kierunek_Lewo            := "KB2_PB_Winda_Tyl",
           Funkcja                  := "KB2_PB_Funkcja",
           Jazda_Prawo              := "KB2_VPB_Winda_Przod",
           Jazda_Lewo               := "KB2_VPB_Winda_Tyl",
           Obrot_Prawo              := "KB2_VPB_Winda_Dol",
           Obrot_Lewo               := "KB2_VPB_Winda_Gora");
NETWORK
TITLE = Lampka kolor zielony str 19
//Lampki wieza sygnalizacyjna
      A     "Zawsze_True";
      =     L 0.0;
      A     L 0.0;
      A     "KB2_Auto_Reczny";
      A     "KB2_M_Bezpieczenstwa_0";
      =     "KB2_Lampa_Kol_Ziel";
      A     L 0.0;
      AN    "KB2_Auto_Reczny";
      A     "KB2_M_Bezpieczenstwa_0";
      =     "KB2_Lampa_Kol_Pom";
      A     L 0.0;
      A     "KB2_Blada_Lini";
      =     "KB2_Lampa_Kol_Czerw";
END_FUNCTION

FUNCTION "Auto_Reczny_Buff" : VOID	// FC 15
VERSION : 0.1
VAR_TEMP
  Temp_Help_1 : BOOL ;
  Temp_Help_2 : BOOL ;
END_VAR
BEGIN
NETWORK
TITLE =
//Ten network celowo jest wolny
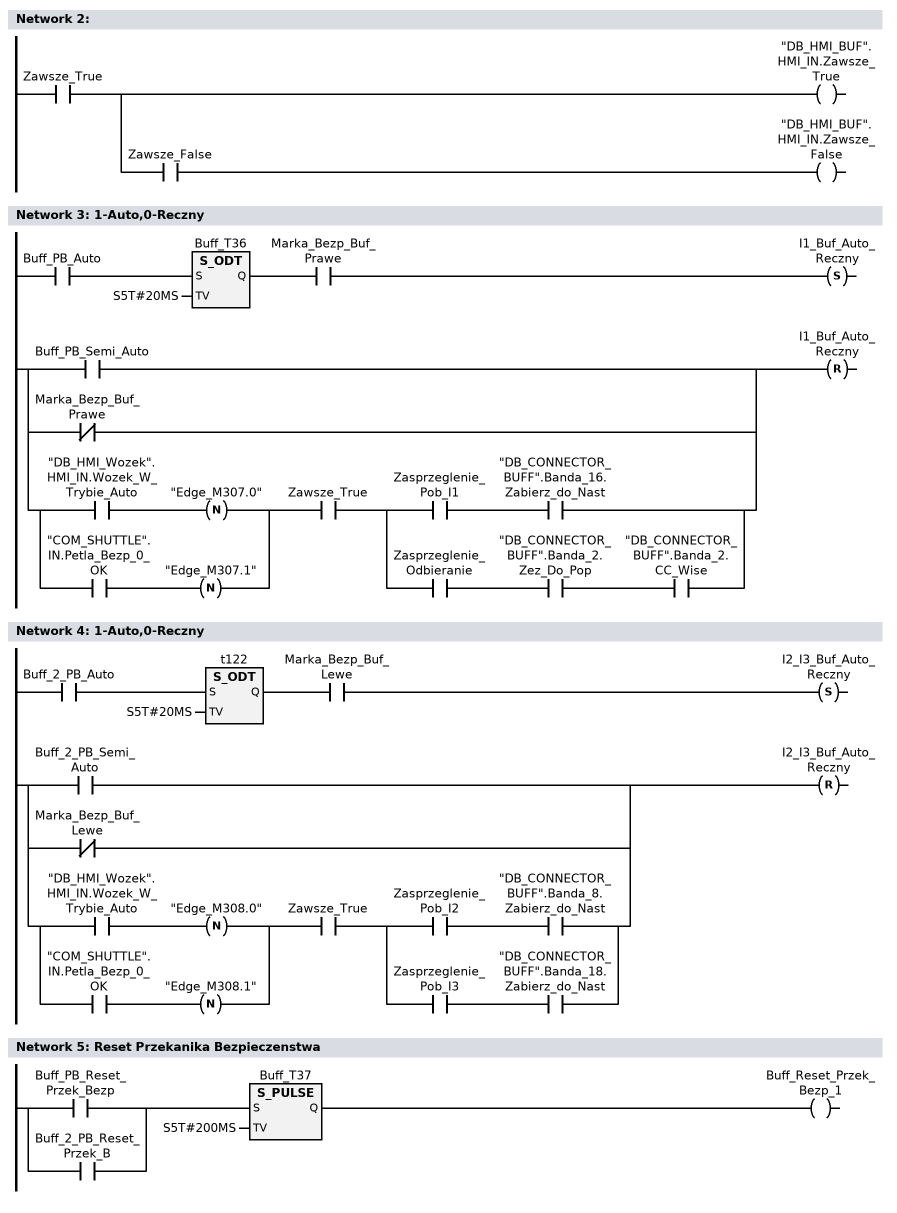
NETWORK
TITLE =
//Dla bufforow
      A     "Zawsze_True";
      =     L 1.0;
      A     L 1.0;
      BLD   102;
      =     "DB_HMI_BUF".HMI_IN.Zawsze_True;
      A     L 1.0;
      A     "Zawsze_False";
      =     "DB_HMI_BUF".HMI_IN.Zawsze_False;
NETWORK
TITLE = 1-Auto,0-Reczny
//Wybranie trybu auto
      A(;
      A     "Buff_PB_Auto";
      L     S5T#20MS;
      SD    "Buff_T36";
      NOP   0;
      NOP   0;
      NOP   0;
      A     "Buff_T36";
      );
      A     "Marka_Bezp_Buf_Prawe";
      S     "I1_Buf_Auto_Reczny";
      A(;
      O     "Buff_PB_Semi_Auto";
      ON    "Marka_Bezp_Buf_Prawe";
      O(;
      A(;
      A     "DB_HMI_Wozek".HMI_IN.Wozek_W_Trybie_Auto;
      FN    "Edge_M307.0";
      O(;
      A     "COM_SHUTTLE".IN.Petla_Bezp_0_OK;
      FN    "Edge_M307.1";
      );
      );
      A     "Zawsze_True";
      A(;
      A     "Zasprzeglenie_Pob_I1";
      A     "DB_CONNECTOR_BUFF".Banda_16.Zabierz_do_Nast;
      O;
      A     "Zasprzeglenie_Odbieranie";
      A     "DB_CONNECTOR_BUFF".Banda_2.Zez_Do_Pop;
      A     "DB_CONNECTOR_BUFF".Banda_2.CC_Wise;
      );
      );
      );
      R     "I1_Buf_Auto_Reczny";
      NOP   0;
NETWORK
TITLE = 1-Auto,0-Reczny
//Wybranie trybu auto
      A(;
      A     "Buff_2_PB_Auto";
      L     S5T#20MS;
      SD    "t122";
      NOP   0;
      NOP   0;
      NOP   0;
      A     "t122";
      );
      A     "Marka_Bezp_Buf_Lewe";
      S     "I2_I3_Buf_Auto_Reczny";
      A(;
      O     "Buff_2_PB_Semi_Auto";
      ON    "Marka_Bezp_Buf_Lewe";
      O(;
      A(;
      A     "DB_HMI_Wozek".HMI_IN.Wozek_W_Trybie_Auto;
      FN    "Edge_M308.0";
      O(;
      A     "COM_SHUTTLE".IN.Petla_Bezp_0_OK;
      FN    "Edge_M308.1";
      );
      );
      A     "Zawsze_True";
      A(;
      A     "Zasprzeglenie_Pob_I2";
      A     "DB_CONNECTOR_BUFF".Banda_8.Zabierz_do_Nast;
      O;
      A     "Zasprzeglenie_Pob_I3";
      A     "DB_CONNECTOR_BUFF".Banda_18.Zabierz_do_Nast;
      );
      );
      );
      R     "I2_I3_Buf_Auto_Reczny";
      NOP   0;
NETWORK
TITLE = Reset Przekanika Bezpieczenstwa
//Reset przekanika bezpieczenstwa. Wspolny dla obu stanowisk
//
      A(;
      O     "Buff_PB_Reset_Przek_Bezp";
      O     "Buff_2_PB_Reset_Przek_B";
      );
      L     S5T#200MS;
      SP    "Buff_T37";
      NOP   0;
      NOP   0;
      NOP   0;
      A     "Buff_T37";
      =     "Buff_Reset_Przek_Bezp_1";
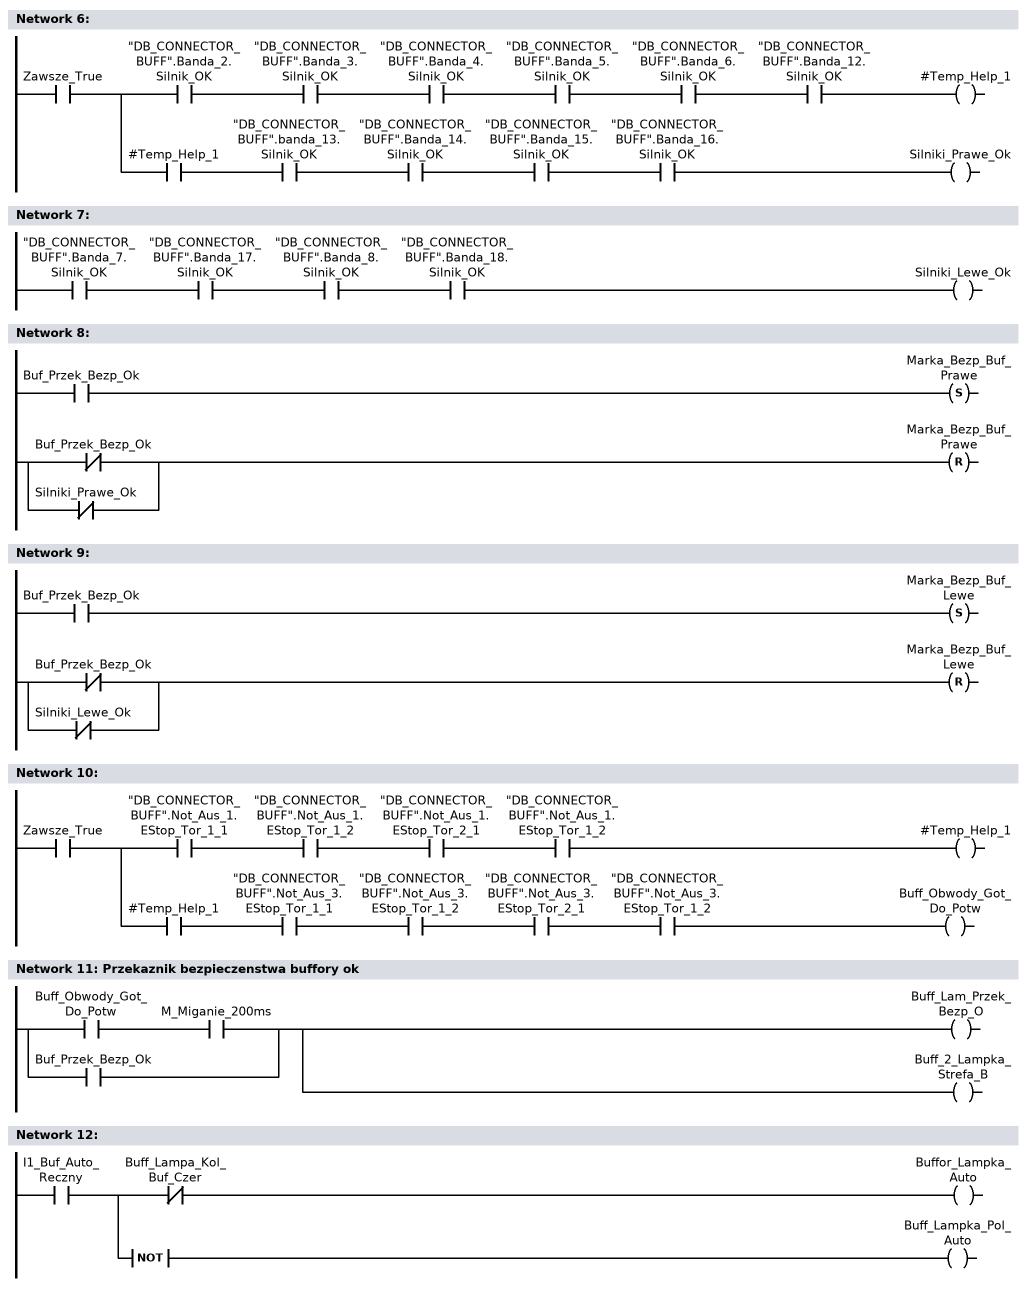
NETWORK
TITLE =
//sprawdz czy silnik sa ok
      A     "Zawsze_True";
      =     L 1.0;
      A     L 1.0;
      A     "DB_CONNECTOR_BUFF".Banda_2.Silnik_OK;
      A     "DB_CONNECTOR_BUFF".Banda_3.Silnik_OK;
      A     "DB_CONNECTOR_BUFF".Banda_4.Silnik_OK;
      A     "DB_CONNECTOR_BUFF".Banda_5.Silnik_OK;
      A     "DB_CONNECTOR_BUFF".Banda_6.Silnik_OK;
      A     "DB_CONNECTOR_BUFF".Banda_12.Silnik_OK;
      =     #Temp_Help_1;
      A     L 1.0;
      A     #Temp_Help_1;
      A     "DB_CONNECTOR_BUFF".banda_13.Silnik_OK;
      A     "DB_CONNECTOR_BUFF".Banda_14.Silnik_OK;
      A     "DB_CONNECTOR_BUFF".Banda_15.Silnik_OK;
      A     "DB_CONNECTOR_BUFF".Banda_16.Silnik_OK;
      =     "Silniki_Prawe_Ok";
NETWORK
TITLE =
//Silniki lewe ok
      A     "DB_CONNECTOR_BUFF".Banda_7.Silnik_OK;
      A     "DB_CONNECTOR_BUFF".Banda_17.Silnik_OK;
      A     "DB_CONNECTOR_BUFF".Banda_8.Silnik_OK;
      A     "DB_CONNECTOR_BUFF".Banda_18.Silnik_OK;
      =     "Silniki_Lewe_Ok";
NETWORK
TITLE =
//Sprawdzenie marki bezpieczenstwa
      A     "Buf_Przek_Bezp_Ok";
      S     "Marka_Bezp_Buf_Prawe";
      A(;
      ON    "Buf_Przek_Bezp_Ok";
      ON    "Silniki_Prawe_Ok";
      );
      R     "Marka_Bezp_Buf_Prawe";
      NOP   0;
NETWORK
TITLE =
//Sprawdzenie marki bezpieczenstwa lewej strony
      A     "Buf_Przek_Bezp_Ok";
      S     "Marka_Bezp_Buf_Lewe";
      A(;
      ON    "Buf_Przek_Bezp_Ok";
      ON    "Silniki_Lewe_Ok";
      );
      R     "Marka_Bezp_Buf_Lewe";
      NOP   0;
NETWORK
TITLE =
//Zprawdzenie czy wszystkie styki Not-Aus ok.
      A     "Zawsze_True";
      =     L 1.0;
      A     L 1.0;
      A     "DB_CONNECTOR_BUFF".Not_Aus_1.EStop_Tor_1_1;
      A     "DB_CONNECTOR_BUFF".Not_Aus_1.EStop_Tor_1_2;
      A     "DB_CONNECTOR_BUFF".Not_Aus_1.EStop_Tor_2_1;
      A     "DB_CONNECTOR_BUFF".Not_Aus_1.EStop_Tor_1_2;
      =     #Temp_Help_1;
      A     L 1.0;
      A     #Temp_Help_1;
      A     "DB_CONNECTOR_BUFF".Not_Aus_3.EStop_Tor_1_1;
      A     "DB_CONNECTOR_BUFF".Not_Aus_3.EStop_Tor_1_2;
      A     "DB_CONNECTOR_BUFF".Not_Aus_3.EStop_Tor_2_1;
      A     "DB_CONNECTOR_BUFF".Not_Aus_3.EStop_Tor_1_2;
      =     "Buff_Obwody_Got_Do_Potw";
NETWORK
TITLE = Przekaznik bezpieczenstwa buffory ok
//Miganie lampki resetu gdy not-aus ok ,a przekaznik bezpieczenstwa jeszcze nie 
//wysterowany
      A     "Buff_Obwody_Got_Do_Potw";
      A     "M_Miganie_200ms";
      O     "Buf_Przek_Bezp_Ok";
      =     "Buff_Lam_Przek_Bezp_O";
      =     "Buff_2_Lampka_Strefa_B";
NETWORK
TITLE =
//Lampki bufor prawy
      A     "I1_Buf_Auto_Reczny";
      =     L 1.0;
      A     L 1.0;
      AN    "Buff_Lampa_Kol_Buf_Czer";
      =     "Buffor_Lampka_Auto";
      A     L 1.0;
      NOT;
      =     "Buff_Lampka_Pol_Auto";
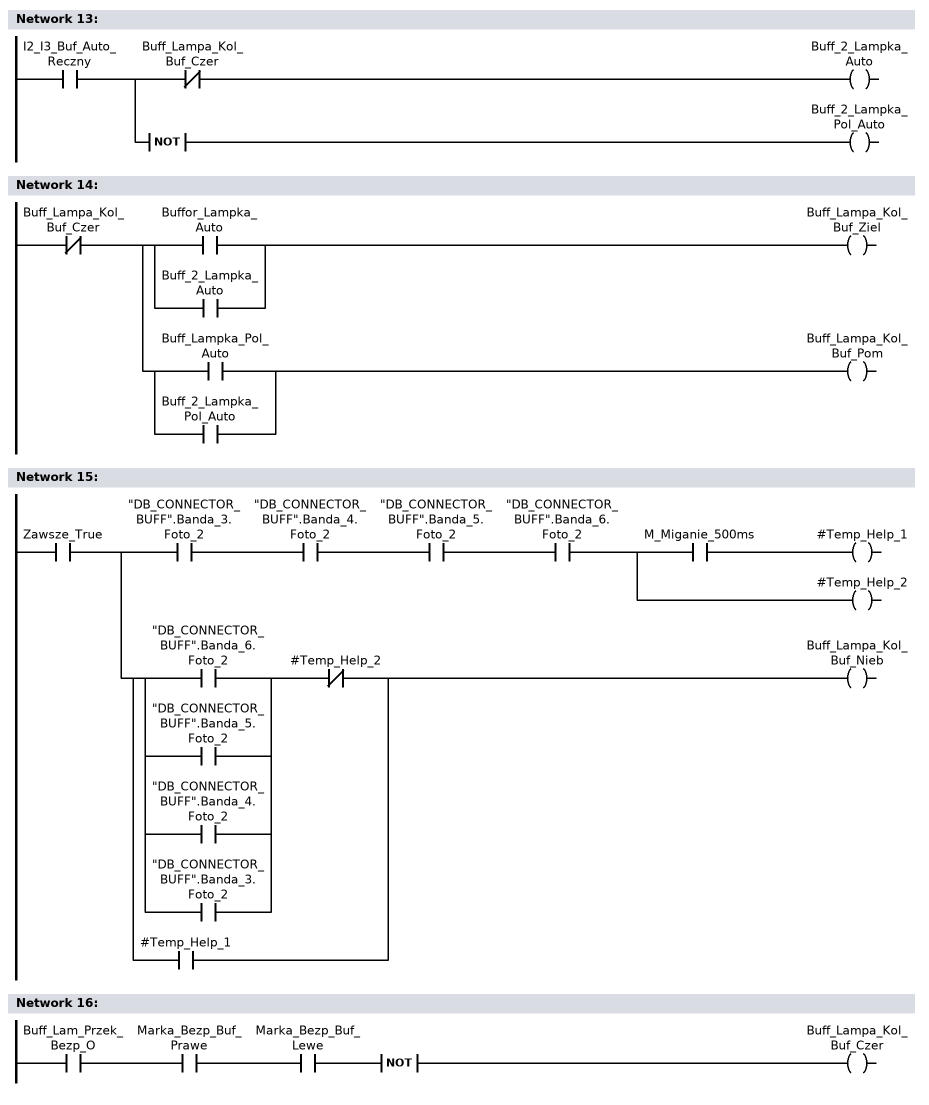
NETWORK
TITLE =
//Lampki bufor prawy
      A     "I2_I3_Buf_Auto_Reczny";
      =     L 1.0;
      A     L 1.0;
      AN    "Buff_Lampa_Kol_Buf_Czer";
      =     "Buff_2_Lampka_Auto";
      A     L 1.0;
      NOT;
      =     "Buff_2_Lampka_Pol_Auto";
NETWORK
TITLE =
//Wieza sygnalizacyjna lampka zolta lub zielona
      AN    "Buff_Lampa_Kol_Buf_Czer";
      =     L 1.0;
      A     L 1.0;
      A(;
      O     "Buffor_Lampka_Auto";
      O     "Buff_2_Lampka_Auto";
      );
      =     "Buff_Lampa_Kol_Buf_Ziel";
      A     L 1.0;
      A(;
      O     "Buff_Lampka_Pol_Auto";
      O     "Buff_2_Lampka_Pol_Auto";
      );
      =     "Buff_Lampa_Kol_Buf_Pom";
NETWORK
TITLE =
//Lampka niebieska informacja ze paleta jest na podajniku
      A     "Zawsze_True";
      =     L 1.0;
      A     L 1.0;
      A     "DB_CONNECTOR_BUFF".Banda_3.Foto_2;
      A     "DB_CONNECTOR_BUFF".Banda_4.Foto_2;
      A     "DB_CONNECTOR_BUFF".Banda_5.Foto_2;
      A     "DB_CONNECTOR_BUFF".Banda_6.Foto_2;
      =     L 1.1;
      A     L 1.1;
      A     "M_Miganie_500ms";
      =     #Temp_Help_1;
      A     L 1.1;
      BLD   102;
      =     #Temp_Help_2;
      A     L 1.0;
      A(;
      A(;
      O     "DB_CONNECTOR_BUFF".Banda_6.Foto_2;
      O     "DB_CONNECTOR_BUFF".Banda_5.Foto_2;
      O     "DB_CONNECTOR_BUFF".Banda_4.Foto_2;
      O     "DB_CONNECTOR_BUFF".Banda_3.Foto_2;
      );
      AN    #Temp_Help_2;
      O     #Temp_Help_1;
      );
      =     "Buff_Lampa_Kol_Buf_Nieb";
NETWORK
TITLE =
//Bufor lampka czerwona
//
      A     "Buff_Lam_Przek_Bezp_O";
      A     "Marka_Bezp_Buf_Prawe";
      A     "Marka_Bezp_Buf_Lewe";
      NOT;
      =     "Buff_Lampa_Kol_Buf_Czer";
END_FUNCTION

FUNCTION "Przypis_Wejsc_KB1" : VOID	// FC 22
//Pobranie z bloku db stanu wejsc sieci asi i przyporzadkowanie do odpowiedniego 
//urzadzenia lini.
//
//Uwaga fotokomorki obrotnicy
//
AUTHOR : Kng
NAME : KB1
VERSION : 0.1
VAR_TEMP
  Help_Bit_1 : BOOL ;
  Help_Bit_2 : BOOL ;
  Help_Word_1 : INT ;
  Help_Word_2 : INT ;
END_VAR
BEGIN
NETWORK
TITLE =
//Ten network celowo jest wolny
NETWORK
TITLE = Silnik ok
//Banda Adres 1 (Wirtualna) bo nalezy do segberta
NETWORK
TITLE = Silnik ok
//Banda Adres 2 (tasma obrotnica)
      A     "DB_ASI_Prosty_Odczyt_KB1".Adres_2_bit_0;
      =     "DB_CONECTOR_KB1".Tasma_Obrotnica.Silnik_OK;
      A     "DB_ASI_Prosty_Odczyt_KB1".Adres_2_bit_1;
      =     "DB_CONECTOR_KB1".Tasma_Obrotnica.Rezerwa_Silnik;
//      A     "DB_ASI_Prosty_Odczyt_KB1".Adres_2_bit_2
      A     "KB1_Obr_Foto_2";
      =     "DB_CONECTOR_KB1".Tasma_Obrotnica.Foto_2;
      A     "KB1_Obr_Foto_1";
//      A     "DB_ASI_Prosty_Odczyt_KB1".Adres_2_bit_3
      =     "DB_CONECTOR_KB1".Tasma_Obrotnica.Foto_1;
NETWORK
TITLE = Silnik ok
//Banda Adres 3
      A     "DB_ASI_Prosty_Odczyt_KB1".Adres_3_bit_0;
      =     "DB_CONECTOR_KB1".Winda.Silnik_OK;
      A     "DB_ASI_Prosty_Odczyt_KB1".Adres_3_bit_1;
      =     "DB_CONECTOR_KB1".Winda.Rezerwa_Silnik;
      A     "DB_ASI_Prosty_Odczyt_KB1".Adres_3_bit_2;
      =     "DB_CONECTOR_KB1".Winda.Foto_1;
      A     "DB_ASI_Prosty_Odczyt_KB1".Adres_3_bit_3;
      =     "DB_CONECTOR_KB1".Winda.Foto_2;
NETWORK
TITLE = Silnik ok
//Banda Adres 4 Silnik Wylot
      A     "DB_ASI_Prosty_Odczyt_KB1".Adres_4_bit_0;
      =     "DB_CONECTOR_KB1".Banda_Wylot_2.Silnik_OK;
      A     "DB_ASI_Prosty_Odczyt_KB1".Adres_4_bit_1;
      =     "DB_CONECTOR_KB1".Banda_Wylot_2.Rezerwa_Silnik;
      A     "DB_ASI_Prosty_Odczyt_KB1".Adres_4_bit_2;
      =     "DB_CONECTOR_KB1".Banda_Wylot_2.Foto_2;
      A     "DB_ASI_Prosty_Odczyt_KB1".Adres_4_bit_3;
      =     "DB_CONECTOR_KB1".Banda_Wylot_2.Foto_1;
NETWORK
TITLE = Silnik ok
//Banda Adres 5 Wirualny (shuttle)
NETWORK
TITLE = Silnik ok
//Obrotnica Adres 9 Wirtualny
NETWORK
TITLE = Silnik ok
//Czujniki Obrotnicy
      A     "DB_ASI_Prosty_Odczyt_KB1".Adres_10_bit_0;
      =     "DB_CONECTOR_KB1".Czujniki_Obr.Czujnik_0_St;
      A     "DB_ASI_Prosty_Odczyt_KB1".Adres_10_bit_1;
      =     "DB_CONECTOR_KB1".Czujniki_Obr.Czujnik_Ham_0_St;
      A     "DB_ASI_Prosty_Odczyt_KB1".Adres_10_bit_2;
      =     "DB_CONECTOR_KB1".Czujniki_Obr.Czujnik_Ham_90_St;
      A     "DB_ASI_Prosty_Odczyt_KB1".Adres_10_bit_3;
      =     "DB_CONECTOR_KB1".Czujniki_Obr.Czujnik_90_St;
NETWORK
TITLE = Silnik ok
//Not-Aus pulpit Adres 20
      A     "DB_ASI_Prosty_Odczyt_KB1".Adres_20_bit_0;
      =     "DB_CONECTOR_KB1".EStop_Pulpit.EStop_Tor_1_1;
      A     "DB_ASI_Prosty_Odczyt_KB1".Adres_20_bit_1;
      =     "DB_CONECTOR_KB1".EStop_Pulpit.EStop_Tor_1_2;
      A     "DB_ASI_Prosty_Odczyt_KB1".Adres_20_bit_2;
      =     "DB_CONECTOR_KB1".EStop_Pulpit.EStop_Tor_2_1;
      A     "DB_ASI_Prosty_Odczyt_KB1".Adres_20_bit_3;
      =     "DB_CONECTOR_KB1".EStop_Pulpit.EStop_Tor_2_2;
NETWORK
TITLE = Silnik ok
//Grzyb bezpieczenstwa Adres 21
      A     "DB_ASI_Prosty_Odczyt_KB1".Adres_21_bit_0;
      =     "DB_CONECTOR_KB1".Estop_Grzyb_Bezp.EStop_Tor_1_1;
      A     "DB_ASI_Prosty_Odczyt_KB1".Adres_21_bit_1;
      =     "DB_CONECTOR_KB1".Estop_Grzyb_Bezp.EStop_Tor_1_2;
      A     "DB_ASI_Prosty_Odczyt_KB1".Adres_21_bit_2;
      =     "DB_CONECTOR_KB1".Estop_Grzyb_Bezp.EStop_Tor_2_1;
      A     "DB_ASI_Prosty_Odczyt_KB1".Adres_21_bit_3;
      =     "DB_CONECTOR_KB1".Estop_Grzyb_Bezp.EStop_Tor_2_2;
NETWORK
TITLE = Silnik ok
//Not-Aus Shuttle Adres 22
      A     "DB_ASI_Prosty_Odczyt_KB1".Adres_22_bit_0;
      =     "DB_CONECTOR_KB1".Estop_Shuttle.EStop_Tor_1_1;
      A     "DB_ASI_Prosty_Odczyt_KB1".Adres_22_bit_1;
      =     "DB_CONECTOR_KB1".Estop_Shuttle.EStop_Tor_1_2;
      A     "DB_ASI_Prosty_Odczyt_KB1".Adres_22_bit_2;
      =     "DB_CONECTOR_KB1".Estop_Shuttle.EStop_Tor_2_1;
      A     "DB_ASI_Prosty_Odczyt_KB1".Adres_22_bit_3;
      =     "DB_CONECTOR_KB1".Estop_Shuttle.EStop_Tor_2_2;
END_FUNCTION

FUNCTION "Przypis_Wyjsc_KB1" : VOID	// FC 23
AUTHOR : Kng
NAME : KB1
VERSION : 0.1
VAR_TEMP
  Temp_Word_1 : INT ;
  Help_Bit_1 : BOOL ;
  Help_Predkosc : REAL ;
END_VAR
BEGIN
NETWORK
TITLE =
//Ten Network celowo jest wolny
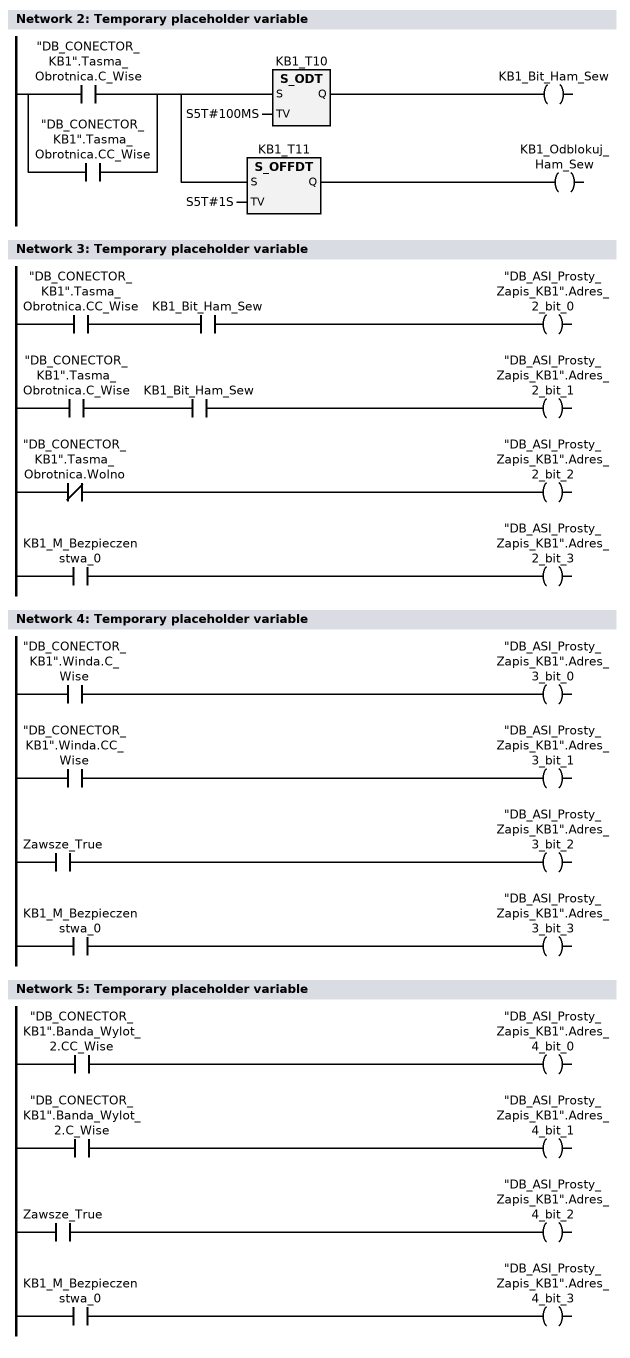
NETWORK
TITLE = Temporary placeholder variable
//Banda Segbert Adres 1 (Wirtualny)
      O     "DB_CONECTOR_KB1".Tasma_Obrotnica.C_Wise;
      O     "DB_CONECTOR_KB1".Tasma_Obrotnica.CC_Wise;
      =     L 8.0;
      A     L 8.0;
      L     S5T#100MS;
      SD    "KB1_T10";
      NOP   0;
      NOP   0;
      NOP   0;
      A     "KB1_T10";
      =     "KB1_Bit_Ham_Sew";
      A     L 8.0;
      L     S5T#1S;
      SF    "KB1_T11";
      NOP   0;
      NOP   0;
      NOP   0;
      A     "KB1_T11";
      =     "KB1_Odblokuj_Ham_Sew";
NETWORK
TITLE = Temporary placeholder variable
//Banda Obrotnica Adres 2
//****************ClockWise*******************
      A     "DB_CONECTOR_KB1".Tasma_Obrotnica.CC_Wise;	//C_Wise
      A     "KB1_Bit_Ham_Sew";
      =     "DB_ASI_Prosty_Zapis_KB1".Adres_2_bit_0;
//****************CounterClockWise************
      A     "DB_CONECTOR_KB1".Tasma_Obrotnica.C_Wise;
      A     "KB1_Bit_Ham_Sew";
      =     "DB_ASI_Prosty_Zapis_KB1".Adres_2_bit_1;	//CC_Wise
//****************Wolno***********************
      AN    "DB_CONECTOR_KB1".Tasma_Obrotnica.Wolno;
      =     "DB_ASI_Prosty_Zapis_KB1".Adres_2_bit_2;	//Wolno
//****************Bit_Bezpieczenstwa**********
      A     "KB1_M_Bezpieczenstwa_0";	//Safety
      =     "DB_ASI_Prosty_Zapis_KB1".Adres_2_bit_3;
NETWORK
TITLE = Temporary placeholder variable
//Winda  Adres 3
//****************ClockWise*******************
      A     "DB_CONECTOR_KB1".Winda.C_Wise;	//C_Wise
      =     "DB_ASI_Prosty_Zapis_KB1".Adres_3_bit_0;
//****************CounterClockWise************
      A     "DB_CONECTOR_KB1".Winda.CC_Wise;
      =     "DB_ASI_Prosty_Zapis_KB1".Adres_3_bit_1;	//CC_Wise
//****************Wolno***********************
      A     "Zawsze_True";
      =     "DB_ASI_Prosty_Zapis_KB1".Adres_3_bit_2;	//Wolno
//****************Bit_Bezpieczenstwa**********
      A     "KB1_M_Bezpieczenstwa_0";
      =     "DB_ASI_Prosty_Zapis_KB1".Adres_3_bit_3;
NETWORK
TITLE = Temporary placeholder variable
//Banda Wylot 2
//****************ClockWise*******************
      A     "DB_CONECTOR_KB1".Banda_Wylot_2.CC_Wise;	//C_Wise
      =     "DB_ASI_Prosty_Zapis_KB1".Adres_4_bit_0;
//****************CounterClockWise************
      A     "DB_CONECTOR_KB1".Banda_Wylot_2.C_Wise;
      =     "DB_ASI_Prosty_Zapis_KB1".Adres_4_bit_1;	//CC_Wise
//****************Wolno***********************
      A     "Zawsze_True";
      =     "DB_ASI_Prosty_Zapis_KB1".Adres_4_bit_2;	//Wolno
//****************Bit_Bezpieczenstwa**********
      A     "KB1_M_Bezpieczenstwa_0";	//Safety
      =     "DB_ASI_Prosty_Zapis_KB1".Adres_4_bit_3;
NETWORK
TITLE = Temporary placeholder variable
//Shuttle adres  5 (Wirtualny) 
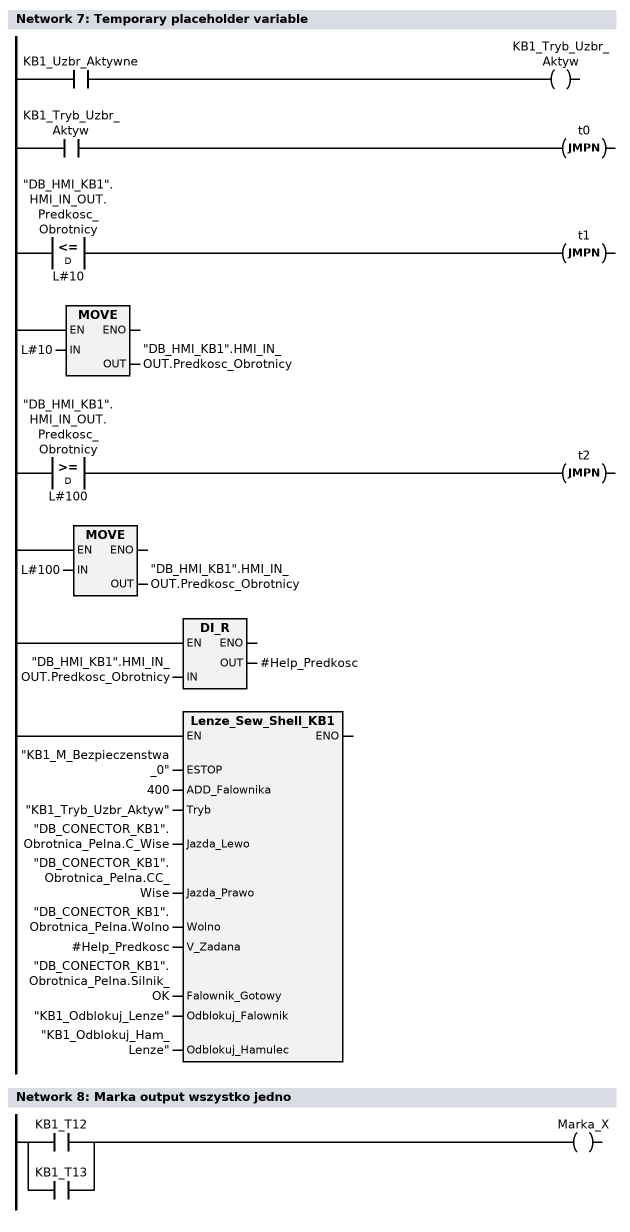
NETWORK
TITLE = Temporary placeholder variable
//Obrotnica Adres  9(Wirtualny)
// Dopasownie predkosci niskiej i wysokiej
      A     "KB1_Uzbr_Aktywne";
      =     "KB1_Tryb_Uzbr_Aktyw";
//************Przypisanie predkosci z panela*************
      A     "KB1_Tryb_Uzbr_Aktyw";
      JCN   t0;
//***Sprawdzenie czy predkosc nie jest za mala
      L     "DB_HMI_KB1".HMI_IN_OUT.Predkosc_Obrotnicy;
      L     L#10;
      <=D;
      JCN   t1;
      L     L#10;
      T     "DB_HMI_KB1".HMI_IN_OUT.Predkosc_Obrotnicy;
t1:   NOP   0;
//***Sprawdzenie czy predkosc nie jest za duza
      L     "DB_HMI_KB1".HMI_IN_OUT.Predkosc_Obrotnicy;
      L     L#100;
      >=D;
      JCN   t2;
      L     L#100;
      T     "DB_HMI_KB1".HMI_IN_OUT.Predkosc_Obrotnicy;
t2:   NOP   0;
//****Zamiana na real
t0:   NOP   0;
      L     "DB_HMI_KB1".HMI_IN_OUT.Predkosc_Obrotnicy;
      DTR;
      T     #Help_Predkosc;
//***Obsluga obrotnicy
      CALL  "Lenze_Sew_Shell_KB1" (
           ESTOP                    := "KB1_M_Bezpieczenstwa_0",
           ADD_Falownika            := 400,
           Tryb                     := "KB1_Tryb_Uzbr_Aktyw",
           Jazda_Lewo               := "DB_CONECTOR_KB1".Obrotnica_Pelna.C_Wise,
           Jazda_Prawo              := "DB_CONECTOR_KB1".Obrotnica_Pelna.CC_Wise,
           Wolno                    := "DB_CONECTOR_KB1".Obrotnica_Pelna.Wolno,
           V_Zadana                 := #Help_Predkosc,
           Falownik_Gotowy          := "DB_CONECTOR_KB1".Obrotnica_Pelna.Silnik_OK,
           Odblokuj_Falownik        := "KB1_Odblokuj_Lenze",
           Odblokuj_Hamulec         := "KB1_Odblokuj_Ham_Lenze");
NETWORK
TITLE = Marka output wszystko jedno
//Wpisz Timmer do rejestru
      O     "KB1_T12";
      O     "KB1_T13";
      =     "Marka_X";
END_FUNCTION

FUNCTION "Przypis_Wejsc_KB2" : VOID	// FC 24
//Pobranie z bloku db stanu wejsc sieci asi i przyporzadkowanie do odpowiedniego 
//urzadzenia lini.
//
//
AUTHOR : Kng
NAME : KB2
VERSION : 0.1
VAR_TEMP
  Help_Bit_1 : BOOL ;
  Help_Bit_2 : BOOL ;
  Help_Word_1 : INT ;
  Help_Word_2 : INT ;
END_VAR
BEGIN
NETWORK
TITLE =
//Ten network celowo jest wolny
NETWORK
TITLE = Silnik ok
//Banda Adres 1 (Wirtualna) bo nalezy do segberta
NETWORK
TITLE = Silnik ok
//Banda Adres 2 (tasma obrotnica)
      A     "DB_ASI_Prosty_Odczyt_KB2".Adres_2_bit_0;
      =     "DB_CONECTOR_KB2".Tasma_Obrotnica.Silnik_OK;
      A     "DB_ASI_Prosty_Odczyt_KB2".Adres_2_bit_1;
      =     "DB_CONECTOR_KB2".Tasma_Obrotnica.Rezerwa_Silnik;
//      A     "DB_ASI_Prosty_Odczyt_KB2".Adres_2_bit_2
      A     "KB2_Obr_Foto_2";
      =     "DB_CONECTOR_KB2".Tasma_Obrotnica.Foto_2;
      A     "KB2_Obr_Foto_1";
//      A     "DB_ASI_Prosty_Odczyt_KB2".Adres_2_bit_3
      =     "DB_CONECTOR_KB2".Tasma_Obrotnica.Foto_1;
NETWORK
TITLE = Silnik ok
//Banda Adres 3
      A     "DB_ASI_Prosty_Odczyt_KB2".Adres_3_bit_0;
      =     "DB_CONECTOR_KB2".Winda.Silnik_OK;
      A     "DB_ASI_Prosty_Odczyt_KB2".Adres_3_bit_1;
      =     "DB_CONECTOR_KB2".Winda.Rezerwa_Silnik;
      A     "DB_ASI_Prosty_Odczyt_KB2".Adres_3_bit_2;
      =     "DB_CONECTOR_KB2".Winda.Foto_1;
      A     "DB_ASI_Prosty_Odczyt_KB2".Adres_3_bit_3;
      =     "DB_CONECTOR_KB2".Winda.Foto_2;
NETWORK
TITLE = Silnik ok
//Banda Adres 4 Silnik Wylot
      A     "DB_ASI_Prosty_Odczyt_KB2".Adres_4_bit_0;
      =     "DB_CONECTOR_KB2".Banda_Wylot_2.Silnik_OK;
      A     "DB_ASI_Prosty_Odczyt_KB2".Adres_4_bit_1;
      =     "DB_CONECTOR_KB2".Banda_Wylot_2.Rezerwa_Silnik;
      A     "DB_ASI_Prosty_Odczyt_KB2".Adres_4_bit_2;
      =     "DB_CONECTOR_KB2".Banda_Wylot_2.Foto_2;
      A     "DB_ASI_Prosty_Odczyt_KB2".Adres_4_bit_3;
      =     "DB_CONECTOR_KB2".Banda_Wylot_2.Foto_1;
NETWORK
TITLE = Silnik ok
//Banda Adres 5 Wirualny (shuttle)
NETWORK
TITLE = Silnik ok
//Obrotnica Adres 9 Wirtualny
NETWORK
TITLE = Silnik ok
//Czujniki Obrotnicy
      A     "DB_ASI_Prosty_Odczyt_KB2".Adres_10_bit_0;
      =     "DB_CONECTOR_KB2".Czujniki_Obr.Czujnik_0_St;
      A     "DB_ASI_Prosty_Odczyt_KB2".Adres_10_bit_1;
      =     "DB_CONECTOR_KB2".Czujniki_Obr.Czujnik_Ham_0_St;
      A     "DB_ASI_Prosty_Odczyt_KB2".Adres_10_bit_2;
      =     "DB_CONECTOR_KB2".Czujniki_Obr.Czujnik_Ham_90_St;
      A     "DB_ASI_Prosty_Odczyt_KB2".Adres_10_bit_3;
      =     "DB_CONECTOR_KB2".Czujniki_Obr.Czujnik_90_St;
NETWORK
TITLE = Silnik ok
//Not-Aus pulpit Adres 20
      A     "DB_ASI_Prosty_Odczyt_KB2".Adres_20_bit_0;
      =     "DB_CONECTOR_KB2".EStop_Pulpit.EStop_Tor_1_1;
      A     "DB_ASI_Prosty_Odczyt_KB2".Adres_20_bit_1;
      =     "DB_CONECTOR_KB2".EStop_Pulpit.EStop_Tor_1_2;
      A     "DB_ASI_Prosty_Odczyt_KB2".Adres_20_bit_2;
      =     "DB_CONECTOR_KB2".EStop_Pulpit.EStop_Tor_2_1;
      A     "DB_ASI_Prosty_Odczyt_KB2".Adres_20_bit_3;
      =     "DB_CONECTOR_KB2".EStop_Pulpit.EStop_Tor_2_2;
NETWORK
TITLE = Silnik ok
//Grzyb bezpieczenstwa Adres 21
      A     "DB_ASI_Prosty_Odczyt_KB2".Adres_21_bit_0;
      =     "DB_CONECTOR_KB2".Estop_Grzyb_Bezp.EStop_Tor_1_1;
      A     "DB_ASI_Prosty_Odczyt_KB2".Adres_21_bit_1;
      =     "DB_CONECTOR_KB2".Estop_Grzyb_Bezp.EStop_Tor_1_2;
      A     "DB_ASI_Prosty_Odczyt_KB2".Adres_21_bit_2;
      =     "DB_CONECTOR_KB2".Estop_Grzyb_Bezp.EStop_Tor_2_1;
      A     "DB_ASI_Prosty_Odczyt_KB2".Adres_21_bit_3;
      =     "DB_CONECTOR_KB2".Estop_Grzyb_Bezp.EStop_Tor_2_2;
NETWORK
TITLE = Silnik ok
//Not-Aus Shuttle Adres 22
      A     "DB_ASI_Prosty_Odczyt_KB2".Adres_22_bit_0;
      =     "DB_CONECTOR_KB2".Estop_Shuttle.EStop_Tor_1_1;
      A     "DB_ASI_Prosty_Odczyt_KB2".Adres_22_bit_1;
      =     "DB_CONECTOR_KB2".Estop_Shuttle.EStop_Tor_1_2;
      A     "DB_ASI_Prosty_Odczyt_KB2".Adres_22_bit_2;
      =     "DB_CONECTOR_KB2".Estop_Shuttle.EStop_Tor_2_1;
      A     "DB_ASI_Prosty_Odczyt_KB2".Adres_22_bit_3;
      =     "DB_CONECTOR_KB2".Estop_Shuttle.EStop_Tor_2_2;
END_FUNCTION

FUNCTION "Przypis_Wyjsc_KB2" : VOID	// FC 25
AUTHOR : Kng
NAME : KB2
VERSION : 0.1
VAR_TEMP
  Temp_Word_1 : INT ;
  Help_Bit_1 : BOOL ;
  Help_Predkosc : REAL ;
END_VAR
BEGIN
NETWORK
TITLE =
//Ten Network celowo jest wolny
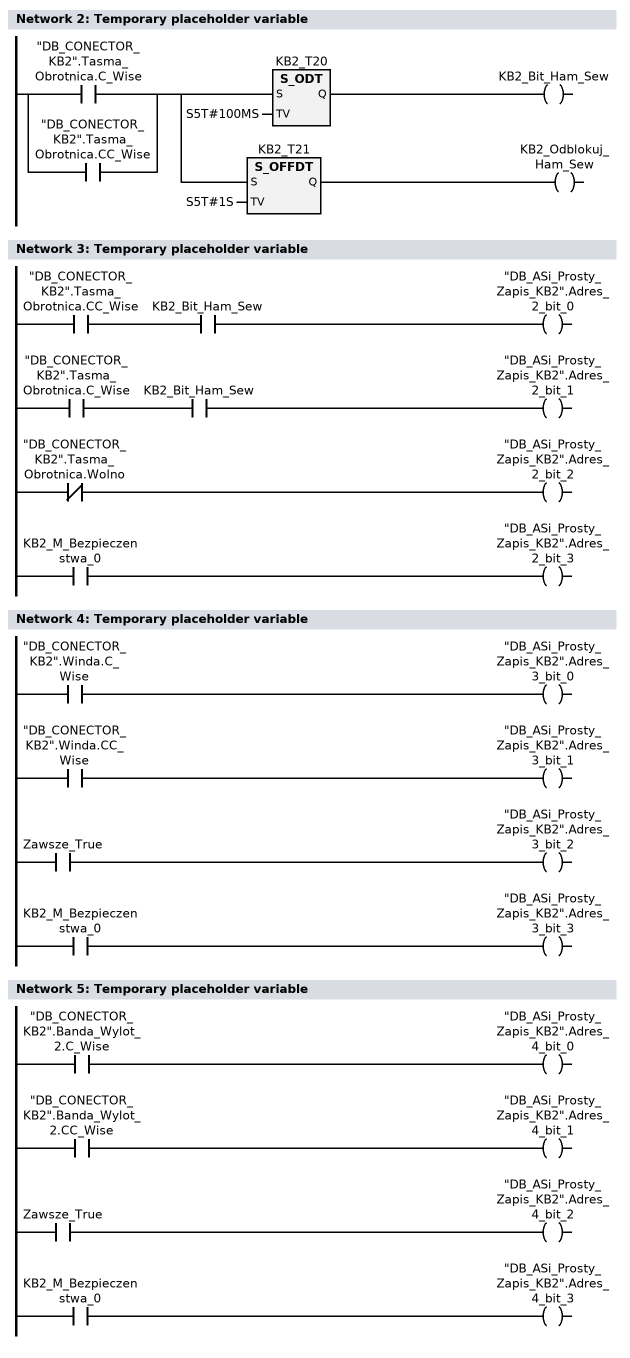
NETWORK
TITLE = Temporary placeholder variable
//Banda Segbert Adres 1 (Wirtualny)
      O     "DB_CONECTOR_KB2".Tasma_Obrotnica.C_Wise;
      O     "DB_CONECTOR_KB2".Tasma_Obrotnica.CC_Wise;
      =     L 8.0;
      A     L 8.0;
      L     S5T#100MS;
      SD    "KB2_T20";
      NOP   0;
      NOP   0;
      NOP   0;
      A     "KB2_T20";
      =     "KB2_Bit_Ham_Sew";
      A     L 8.0;
      L     S5T#1S;
      SF    "KB2_T21";
      NOP   0;
      NOP   0;
      NOP   0;
      A     "KB2_T21";
      =     "KB2_Odblokuj_Ham_Sew";
NETWORK
TITLE = Temporary placeholder variable
//Banda Obrotnica Adres 2
//****************ClockWise*******************
      A     "DB_CONECTOR_KB2".Tasma_Obrotnica.CC_Wise;	//C_Wise
      A     "KB2_Bit_Ham_Sew";
      =     "DB_ASi_Prosty_Zapis_KB2".Adres_2_bit_0;
//****************CounterClockWise************
      A     "DB_CONECTOR_KB2".Tasma_Obrotnica.C_Wise;
      A     "KB2_Bit_Ham_Sew";
      =     "DB_ASi_Prosty_Zapis_KB2".Adres_2_bit_1;	//CC_Wise
//****************Wolno***********************
      AN    "DB_CONECTOR_KB2".Tasma_Obrotnica.Wolno;
      =     "DB_ASi_Prosty_Zapis_KB2".Adres_2_bit_2;	//Wolno
//****************Bit_Bezpieczenstwa**********
      A     "KB2_M_Bezpieczenstwa_0";	//Safety
      =     "DB_ASi_Prosty_Zapis_KB2".Adres_2_bit_3;
NETWORK
TITLE = Temporary placeholder variable
//Winda  Adres 3
//****************ClockWise*******************
      A     "DB_CONECTOR_KB2".Winda.C_Wise;	//C_Wise
      =     "DB_ASi_Prosty_Zapis_KB2".Adres_3_bit_0;
//****************CounterClockWise************
      A     "DB_CONECTOR_KB2".Winda.CC_Wise;
      =     "DB_ASi_Prosty_Zapis_KB2".Adres_3_bit_1;	//CC_Wise
//****************Wolno***********************
      A     "Zawsze_True";
      =     "DB_ASi_Prosty_Zapis_KB2".Adres_3_bit_2;	//Wolno
//****************Bit_Bezpieczenstwa**********
      A     "KB2_M_Bezpieczenstwa_0";
      =     "DB_ASi_Prosty_Zapis_KB2".Adres_3_bit_3;
NETWORK
TITLE = Temporary placeholder variable
//Banda Wylot 2
//****************ClockWise*******************
      A     "DB_CONECTOR_KB2".Banda_Wylot_2.C_Wise;	//C_Wise
      =     "DB_ASi_Prosty_Zapis_KB2".Adres_4_bit_0;
//****************CounterClockWise************
      A     "DB_CONECTOR_KB2".Banda_Wylot_2.CC_Wise;
      =     "DB_ASi_Prosty_Zapis_KB2".Adres_4_bit_1;	//CC_Wise
//****************Wolno***********************
      A     "Zawsze_True";
      =     "DB_ASi_Prosty_Zapis_KB2".Adres_4_bit_2;	//Wolno
//****************Bit_Bezpieczenstwa**********
      A     "KB2_M_Bezpieczenstwa_0";	//Safety
      =     "DB_ASi_Prosty_Zapis_KB2".Adres_4_bit_3;
NETWORK
TITLE = Temporary placeholder variable
//Shuttle adres  5 (Wirtualny) 
